    PROC StoreSlot_P02(num slot, num subType, num toolSel, num lenMM,
                       robtarget arcStart, robtarget arcEnd, robtarget approach, robtarget retract, robtarget trans)
        IF slot = 1 THEN
            P02W01_SubType := subType;
            P02W01_ToolSel := toolSel;
            P02W01_LenMM := lenMM;
            P02W01_ArcStart := arcStart;
            P02W01_ArcEnd := arcEnd;
            P02W01_Approach := approach;
            P02W01_Retract := retract;
            P02W01_Trans := trans;
            P02W01_Used := TRUE;
        ELSEIF slot = 2 THEN
            P02W02_SubType := subType;
            P02W02_ToolSel := toolSel;
            P02W02_LenMM := lenMM;
            P02W02_ArcStart := arcStart;
            P02W02_ArcEnd := arcEnd;
            P02W02_Approach := approach;
            P02W02_Retract := retract;
            P02W02_Trans := trans;
            P02W02_Used := TRUE;
        ELSEIF slot = 3 THEN
            P02W03_SubType := subType;
            P02W03_ToolSel := toolSel;
            P02W03_LenMM := lenMM;
            P02W03_ArcStart := arcStart;
            P02W03_ArcEnd := arcEnd;
            P02W03_Approach := approach;
            P02W03_Retract := retract;
            P02W03_Trans := trans;
            P02W03_Used := TRUE;
        ELSEIF slot = 4 THEN
            P02W04_SubType := subType;
            P02W04_ToolSel := toolSel;
            P02W04_LenMM := lenMM;
            P02W04_ArcStart := arcStart;
            P02W04_ArcEnd := arcEnd;
            P02W04_Approach := approach;
            P02W04_Retract := retract;
            P02W04_Trans := trans;
            P02W04_Used := TRUE;
        ELSEIF slot = 5 THEN
            P02W05_SubType := subType;
            P02W05_ToolSel := toolSel;
            P02W05_LenMM := lenMM;
            P02W05_ArcStart := arcStart;
            P02W05_ArcEnd := arcEnd;
            P02W05_Approach := approach;
            P02W05_Retract := retract;
            P02W05_Trans := trans;
            P02W05_Used := TRUE;
        ELSEIF slot = 6 THEN
            P02W06_SubType := subType;
            P02W06_ToolSel := toolSel;
            P02W06_LenMM := lenMM;
            P02W06_ArcStart := arcStart;
            P02W06_ArcEnd := arcEnd;
            P02W06_Approach := approach;
            P02W06_Retract := retract;
            P02W06_Trans := trans;
            P02W06_Used := TRUE;
        ELSEIF slot = 7 THEN
            P02W07_SubType := subType;
            P02W07_ToolSel := toolSel;
            P02W07_LenMM := lenMM;
            P02W07_ArcStart := arcStart;
            P02W07_ArcEnd := arcEnd;
            P02W07_Approach := approach;
            P02W07_Retract := retract;
            P02W07_Trans := trans;
            P02W07_Used := TRUE;
        ELSEIF slot = 8 THEN
            P02W08_SubType := subType;
            P02W08_ToolSel := toolSel;
            P02W08_LenMM := lenMM;
            P02W08_ArcStart := arcStart;
            P02W08_ArcEnd := arcEnd;
            P02W08_Approach := approach;
            P02W08_Retract := retract;
            P02W08_Trans := trans;
            P02W08_Used := TRUE;
        ELSEIF slot = 9 THEN
            P02W09_SubType := subType;
            P02W09_ToolSel := toolSel;
            P02W09_LenMM := lenMM;
            P02W09_ArcStart := arcStart;
            P02W09_ArcEnd := arcEnd;
            P02W09_Approach := approach;
            P02W09_Retract := retract;
            P02W09_Trans := trans;
            P02W09_Used := TRUE;
        ELSEIF slot = 10 THEN
            P02W10_SubType := subType;
            P02W10_ToolSel := toolSel;
            P02W10_LenMM := lenMM;
            P02W10_ArcStart := arcStart;
            P02W10_ArcEnd := arcEnd;
            P02W10_Approach := approach;
            P02W10_Retract := retract;
            P02W10_Trans := trans;
            P02W10_Used := TRUE;
        ELSEIF slot = 11 THEN
            P02W11_SubType := subType;
            P02W11_ToolSel := toolSel;
            P02W11_LenMM := lenMM;
            P02W11_ArcStart := arcStart;
            P02W11_ArcEnd := arcEnd;
            P02W11_Approach := approach;
            P02W11_Retract := retract;
            P02W11_Trans := trans;
            P02W11_Used := TRUE;
        ELSEIF slot = 12 THEN
            P02W12_SubType := subType;
            P02W12_ToolSel := toolSel;
            P02W12_LenMM := lenMM;
            P02W12_ArcStart := arcStart;
            P02W12_ArcEnd := arcEnd;
            P02W12_Approach := approach;
            P02W12_Retract := retract;
            P02W12_Trans := trans;
            P02W12_Used := TRUE;
        ELSEIF slot = 13 THEN
            P02W13_SubType := subType;
            P02W13_ToolSel := toolSel;
            P02W13_LenMM := lenMM;
            P02W13_ArcStart := arcStart;
            P02W13_ArcEnd := arcEnd;
            P02W13_Approach := approach;
            P02W13_Retract := retract;
            P02W13_Trans := trans;
            P02W13_Used := TRUE;
        ELSEIF slot = 14 THEN
            P02W14_SubType := subType;
            P02W14_ToolSel := toolSel;
            P02W14_LenMM := lenMM;
            P02W14_ArcStart := arcStart;
            P02W14_ArcEnd := arcEnd;
            P02W14_Approach := approach;
            P02W14_Retract := retract;
            P02W14_Trans := trans;
            P02W14_Used := TRUE;
        ELSEIF slot = 15 THEN
            P02W15_SubType := subType;
            P02W15_ToolSel := toolSel;
            P02W15_LenMM := lenMM;
            P02W15_ArcStart := arcStart;
            P02W15_ArcEnd := arcEnd;
            P02W15_Approach := approach;
            P02W15_Retract := retract;
            P02W15_Trans := trans;
            P02W15_Used := TRUE;
        ELSEIF slot = 16 THEN
            P02W16_SubType := subType;
            P02W16_ToolSel := toolSel;
            P02W16_LenMM := lenMM;
            P02W16_ArcStart := arcStart;
            P02W16_ArcEnd := arcEnd;
            P02W16_Approach := approach;
            P02W16_Retract := retract;
            P02W16_Trans := trans;
            P02W16_Used := TRUE;
        ELSEIF slot = 17 THEN
            P02W17_SubType := subType;
            P02W17_ToolSel := toolSel;
            P02W17_LenMM := lenMM;
            P02W17_ArcStart := arcStart;
            P02W17_ArcEnd := arcEnd;
            P02W17_Approach := approach;
            P02W17_Retract := retract;
            P02W17_Trans := trans;
            P02W17_Used := TRUE;
        ELSEIF slot = 18 THEN
            P02W18_SubType := subType;
            P02W18_ToolSel := toolSel;
            P02W18_LenMM := lenMM;
            P02W18_ArcStart := arcStart;
            P02W18_ArcEnd := arcEnd;
            P02W18_Approach := approach;
            P02W18_Retract := retract;
            P02W18_Trans := trans;
            P02W18_Used := TRUE;
        ELSEIF slot = 19 THEN
            P02W19_SubType := subType;
            P02W19_ToolSel := toolSel;
            P02W19_LenMM := lenMM;
            P02W19_ArcStart := arcStart;
            P02W19_ArcEnd := arcEnd;
            P02W19_Approach := approach;
            P02W19_Retract := retract;
            P02W19_Trans := trans;
            P02W19_Used := TRUE;
        ELSEIF slot = 20 THEN
            P02W20_SubType := subType;
            P02W20_ToolSel := toolSel;
            P02W20_LenMM := lenMM;
            P02W20_ArcStart := arcStart;
            P02W20_ArcEnd := arcEnd;
            P02W20_Approach := approach;
            P02W20_Retract := retract;
            P02W20_Trans := trans;
            P02W20_Used := TRUE;
        ELSEIF slot = 21 THEN
            P02W21_SubType := subType;
            P02W21_ToolSel := toolSel;
            P02W21_LenMM := lenMM;
            P02W21_ArcStart := arcStart;
            P02W21_ArcEnd := arcEnd;
            P02W21_Approach := approach;
            P02W21_Retract := retract;
            P02W21_Trans := trans;
            P02W21_Used := TRUE;
        ELSEIF slot = 22 THEN
            P02W22_SubType := subType;
            P02W22_ToolSel := toolSel;
            P02W22_LenMM := lenMM;
            P02W22_ArcStart := arcStart;
            P02W22_ArcEnd := arcEnd;
            P02W22_Approach := approach;
            P02W22_Retract := retract;
            P02W22_Trans := trans;
            P02W22_Used := TRUE;
        ELSEIF slot = 23 THEN
            P02W23_SubType := subType;
            P02W23_ToolSel := toolSel;
            P02W23_LenMM := lenMM;
            P02W23_ArcStart := arcStart;
            P02W23_ArcEnd := arcEnd;
            P02W23_Approach := approach;
            P02W23_Retract := retract;
            P02W23_Trans := trans;
            P02W23_Used := TRUE;
        ELSEIF slot = 24 THEN
            P02W24_SubType := subType;
            P02W24_ToolSel := toolSel;
            P02W24_LenMM := lenMM;
            P02W24_ArcStart := arcStart;
            P02W24_ArcEnd := arcEnd;
            P02W24_Approach := approach;
            P02W24_Retract := retract;
            P02W24_Trans := trans;
            P02W24_Used := TRUE;
        ELSEIF slot = 25 THEN
            P02W25_SubType := subType;
            P02W25_ToolSel := toolSel;
            P02W25_LenMM := lenMM;
            P02W25_ArcStart := arcStart;
            P02W25_ArcEnd := arcEnd;
            P02W25_Approach := approach;
            P02W25_Retract := retract;
            P02W25_Trans := trans;
            P02W25_Used := TRUE;
        ELSEIF slot = 26 THEN
            P02W26_SubType := subType;
            P02W26_ToolSel := toolSel;
            P02W26_LenMM := lenMM;
            P02W26_ArcStart := arcStart;
            P02W26_ArcEnd := arcEnd;
            P02W26_Approach := approach;
            P02W26_Retract := retract;
            P02W26_Trans := trans;
            P02W26_Used := TRUE;
        ELSEIF slot = 27 THEN
            P02W27_SubType := subType;
            P02W27_ToolSel := toolSel;
            P02W27_LenMM := lenMM;
            P02W27_ArcStart := arcStart;
            P02W27_ArcEnd := arcEnd;
            P02W27_Approach := approach;
            P02W27_Retract := retract;
            P02W27_Trans := trans;
            P02W27_Used := TRUE;
        ELSEIF slot = 28 THEN
            P02W28_SubType := subType;
            P02W28_ToolSel := toolSel;
            P02W28_LenMM := lenMM;
            P02W28_ArcStart := arcStart;
            P02W28_ArcEnd := arcEnd;
            P02W28_Approach := approach;
            P02W28_Retract := retract;
            P02W28_Trans := trans;
            P02W28_Used := TRUE;
        ELSEIF slot = 29 THEN
            P02W29_SubType := subType;
            P02W29_ToolSel := toolSel;
            P02W29_LenMM := lenMM;
            P02W29_ArcStart := arcStart;
            P02W29_ArcEnd := arcEnd;
            P02W29_Approach := approach;
            P02W29_Retract := retract;
            P02W29_Trans := trans;
            P02W29_Used := TRUE;
        ELSEIF slot = 30 THEN
            P02W30_SubType := subType;
            P02W30_ToolSel := toolSel;
            P02W30_LenMM := lenMM;
            P02W30_ArcStart := arcStart;
            P02W30_ArcEnd := arcEnd;
            P02W30_Approach := approach;
            P02W30_Retract := retract;
            P02W30_Trans := trans;
            P02W30_Used := TRUE;
        ELSE
            TPWrite "Invalid weld slot.";
        ENDIF
    ENDPROC

    PROC LoadSlot_P02(num slot, VAR bool used, VAR num subType, VAR num toolSel, VAR num lenMM,
                       VAR robtarget arcStart, VAR robtarget arcEnd, VAR robtarget approach, VAR robtarget retract, VAR robtarget trans)
        IF slot = 1 THEN
            used := P02W01_Used;
            subType := P02W01_SubType;
            toolSel := P02W01_ToolSel;
            lenMM := P02W01_LenMM;
            arcStart := P02W01_ArcStart;
            arcEnd := P02W01_ArcEnd;
            approach := P02W01_Approach;
            retract := P02W01_Retract;
            trans := P02W01_Trans;
        ELSEIF slot = 2 THEN
            used := P02W02_Used;
            subType := P02W02_SubType;
            toolSel := P02W02_ToolSel;
            lenMM := P02W02_LenMM;
            arcStart := P02W02_ArcStart;
            arcEnd := P02W02_ArcEnd;
            approach := P02W02_Approach;
            retract := P02W02_Retract;
            trans := P02W02_Trans;
        ELSEIF slot = 3 THEN
            used := P02W03_Used;
            subType := P02W03_SubType;
            toolSel := P02W03_ToolSel;
            lenMM := P02W03_LenMM;
            arcStart := P02W03_ArcStart;
            arcEnd := P02W03_ArcEnd;
            approach := P02W03_Approach;
            retract := P02W03_Retract;
            trans := P02W03_Trans;
        ELSEIF slot = 4 THEN
            used := P02W04_Used;
            subType := P02W04_SubType;
            toolSel := P02W04_ToolSel;
            lenMM := P02W04_LenMM;
            arcStart := P02W04_ArcStart;
            arcEnd := P02W04_ArcEnd;
            approach := P02W04_Approach;
            retract := P02W04_Retract;
            trans := P02W04_Trans;
        ELSEIF slot = 5 THEN
            used := P02W05_Used;
            subType := P02W05_SubType;
            toolSel := P02W05_ToolSel;
            lenMM := P02W05_LenMM;
            arcStart := P02W05_ArcStart;
            arcEnd := P02W05_ArcEnd;
            approach := P02W05_Approach;
            retract := P02W05_Retract;
            trans := P02W05_Trans;
        ELSEIF slot = 6 THEN
            used := P02W06_Used;
            subType := P02W06_SubType;
            toolSel := P02W06_ToolSel;
            lenMM := P02W06_LenMM;
            arcStart := P02W06_ArcStart;
            arcEnd := P02W06_ArcEnd;
            approach := P02W06_Approach;
            retract := P02W06_Retract;
            trans := P02W06_Trans;
        ELSEIF slot = 7 THEN
            used := P02W07_Used;
            subType := P02W07_SubType;
            toolSel := P02W07_ToolSel;
            lenMM := P02W07_LenMM;
            arcStart := P02W07_ArcStart;
            arcEnd := P02W07_ArcEnd;
            approach := P02W07_Approach;
            retract := P02W07_Retract;
            trans := P02W07_Trans;
        ELSEIF slot = 8 THEN
            used := P02W08_Used;
            subType := P02W08_SubType;
            toolSel := P02W08_ToolSel;
            lenMM := P02W08_LenMM;
            arcStart := P02W08_ArcStart;
            arcEnd := P02W08_ArcEnd;
            approach := P02W08_Approach;
            retract := P02W08_Retract;
            trans := P02W08_Trans;
        ELSEIF slot = 9 THEN
            used := P02W09_Used;
            subType := P02W09_SubType;
            toolSel := P02W09_ToolSel;
            lenMM := P02W09_LenMM;
            arcStart := P02W09_ArcStart;
            arcEnd := P02W09_ArcEnd;
            approach := P02W09_Approach;
            retract := P02W09_Retract;
            trans := P02W09_Trans;
        ELSEIF slot = 10 THEN
            used := P02W10_Used;
            subType := P02W10_SubType;
            toolSel := P02W10_ToolSel;
            lenMM := P02W10_LenMM;
            arcStart := P02W10_ArcStart;
            arcEnd := P02W10_ArcEnd;
            approach := P02W10_Approach;
            retract := P02W10_Retract;
            trans := P02W10_Trans;
        ELSEIF slot = 11 THEN
            used := P02W11_Used;
            subType := P02W11_SubType;
            toolSel := P02W11_ToolSel;
            lenMM := P02W11_LenMM;
            arcStart := P02W11_ArcStart;
            arcEnd := P02W11_ArcEnd;
            approach := P02W11_Approach;
            retract := P02W11_Retract;
            trans := P02W11_Trans;
        ELSEIF slot = 12 THEN
            used := P02W12_Used;
            subType := P02W12_SubType;
            toolSel := P02W12_ToolSel;
            lenMM := P02W12_LenMM;
            arcStart := P02W12_ArcStart;
            arcEnd := P02W12_ArcEnd;
            approach := P02W12_Approach;
            retract := P02W12_Retract;
            trans := P02W12_Trans;
        ELSEIF slot = 13 THEN
            used := P02W13_Used;
            subType := P02W13_SubType;
            toolSel := P02W13_ToolSel;
            lenMM := P02W13_LenMM;
            arcStart := P02W13_ArcStart;
            arcEnd := P02W13_ArcEnd;
            approach := P02W13_Approach;
            retract := P02W13_Retract;
            trans := P02W13_Trans;
        ELSEIF slot = 14 THEN
            used := P02W14_Used;
            subType := P02W14_SubType;
            toolSel := P02W14_ToolSel;
            lenMM := P02W14_LenMM;
            arcStart := P02W14_ArcStart;
            arcEnd := P02W14_ArcEnd;
            approach := P02W14_Approach;
            retract := P02W14_Retract;
            trans := P02W14_Trans;
        ELSEIF slot = 15 THEN
            used := P02W15_Used;
            subType := P02W15_SubType;
            toolSel := P02W15_ToolSel;
            lenMM := P02W15_LenMM;
            arcStart := P02W15_ArcStart;
            arcEnd := P02W15_ArcEnd;
            approach := P02W15_Approach;
            retract := P02W15_Retract;
            trans := P02W15_Trans;
        ELSEIF slot = 16 THEN
            used := P02W16_Used;
            subType := P02W16_SubType;
            toolSel := P02W16_ToolSel;
            lenMM := P02W16_LenMM;
            arcStart := P02W16_ArcStart;
            arcEnd := P02W16_ArcEnd;
            approach := P02W16_Approach;
            retract := P02W16_Retract;
            trans := P02W16_Trans;
        ELSEIF slot = 17 THEN
            used := P02W17_Used;
            subType := P02W17_SubType;
            toolSel := P02W17_ToolSel;
            lenMM := P02W17_LenMM;
            arcStart := P02W17_ArcStart;
            arcEnd := P02W17_ArcEnd;
            approach := P02W17_Approach;
            retract := P02W17_Retract;
            trans := P02W17_Trans;
        ELSEIF slot = 18 THEN
            used := P02W18_Used;
            subType := P02W18_SubType;
            toolSel := P02W18_ToolSel;
            lenMM := P02W18_LenMM;
            arcStart := P02W18_ArcStart;
            arcEnd := P02W18_ArcEnd;
            approach := P02W18_Approach;
            retract := P02W18_Retract;
            trans := P02W18_Trans;
        ELSEIF slot = 19 THEN
            used := P02W19_Used;
            subType := P02W19_SubType;
            toolSel := P02W19_ToolSel;
            lenMM := P02W19_LenMM;
            arcStart := P02W19_ArcStart;
            arcEnd := P02W19_ArcEnd;
            approach := P02W19_Approach;
            retract := P02W19_Retract;
            trans := P02W19_Trans;
        ELSEIF slot = 20 THEN
            used := P02W20_Used;
            subType := P02W20_SubType;
            toolSel := P02W20_ToolSel;
            lenMM := P02W20_LenMM;
            arcStart := P02W20_ArcStart;
            arcEnd := P02W20_ArcEnd;
            approach := P02W20_Approach;
            retract := P02W20_Retract;
            trans := P02W20_Trans;
        ELSEIF slot = 21 THEN
            used := P02W21_Used;
            subType := P02W21_SubType;
            toolSel := P02W21_ToolSel;
            lenMM := P02W21_LenMM;
            arcStart := P02W21_ArcStart;
            arcEnd := P02W21_ArcEnd;
            approach := P02W21_Approach;
            retract := P02W21_Retract;
            trans := P02W21_Trans;
        ELSEIF slot = 22 THEN
            used := P02W22_Used;
            subType := P02W22_SubType;
            toolSel := P02W22_ToolSel;
            lenMM := P02W22_LenMM;
            arcStart := P02W22_ArcStart;
            arcEnd := P02W22_ArcEnd;
            approach := P02W22_Approach;
            retract := P02W22_Retract;
            trans := P02W22_Trans;
        ELSEIF slot = 23 THEN
            used := P02W23_Used;
            subType := P02W23_SubType;
            toolSel := P02W23_ToolSel;
            lenMM := P02W23_LenMM;
            arcStart := P02W23_ArcStart;
            arcEnd := P02W23_ArcEnd;
            approach := P02W23_Approach;
            retract := P02W23_Retract;
            trans := P02W23_Trans;
        ELSEIF slot = 24 THEN
            used := P02W24_Used;
            subType := P02W24_SubType;
            toolSel := P02W24_ToolSel;
            lenMM := P02W24_LenMM;
            arcStart := P02W24_ArcStart;
            arcEnd := P02W24_ArcEnd;
            approach := P02W24_Approach;
            retract := P02W24_Retract;
            trans := P02W24_Trans;
        ELSEIF slot = 25 THEN
            used := P02W25_Used;
            subType := P02W25_SubType;
            toolSel := P02W25_ToolSel;
            lenMM := P02W25_LenMM;
            arcStart := P02W25_ArcStart;
            arcEnd := P02W25_ArcEnd;
            approach := P02W25_Approach;
            retract := P02W25_Retract;
            trans := P02W25_Trans;
        ELSEIF slot = 26 THEN
            used := P02W26_Used;
            subType := P02W26_SubType;
            toolSel := P02W26_ToolSel;
            lenMM := P02W26_LenMM;
            arcStart := P02W26_ArcStart;
            arcEnd := P02W26_ArcEnd;
            approach := P02W26_Approach;
            retract := P02W26_Retract;
            trans := P02W26_Trans;
        ELSEIF slot = 27 THEN
            used := P02W27_Used;
            subType := P02W27_SubType;
            toolSel := P02W27_ToolSel;
            lenMM := P02W27_LenMM;
            arcStart := P02W27_ArcStart;
            arcEnd := P02W27_ArcEnd;
            approach := P02W27_Approach;
            retract := P02W27_Retract;
            trans := P02W27_Trans;
        ELSEIF slot = 28 THEN
            used := P02W28_Used;
            subType := P02W28_SubType;
            toolSel := P02W28_ToolSel;
            lenMM := P02W28_LenMM;
            arcStart := P02W28_ArcStart;
            arcEnd := P02W28_ArcEnd;
            approach := P02W28_Approach;
            retract := P02W28_Retract;
            trans := P02W28_Trans;
        ELSEIF slot = 29 THEN
            used := P02W29_Used;
            subType := P02W29_SubType;
            toolSel := P02W29_ToolSel;
            lenMM := P02W29_LenMM;
            arcStart := P02W29_ArcStart;
            arcEnd := P02W29_ArcEnd;
            approach := P02W29_Approach;
            retract := P02W29_Retract;
            trans := P02W29_Trans;
        ELSEIF slot = 30 THEN
            used := P02W30_Used;
            subType := P02W30_SubType;
            toolSel := P02W30_ToolSel;
            lenMM := P02W30_LenMM;
            arcStart := P02W30_ArcStart;
            arcEnd := P02W30_ArcEnd;
            approach := P02W30_Approach;
            retract := P02W30_Retract;
            trans := P02W30_Trans;
        ELSE
            used := FALSE;
        ENDIF
    ENDPROC

    PROC ClearSlot_P02(num slot)
        IF slot = 1 THEN
            P02W01_Used := FALSE;
            P02W01_SubType := 0;
            P02W01_ToolSel := 0;
            P02W01_LenMM := 0;
            P02W01_ArcStart := [[0,0,0],[1,0,0,0],[0,0,0,0],[9E9,9E9,9E9,9E9,9E9,9E9]];
            P02W01_ArcEnd := [[0,0,0],[1,0,0,0],[0,0,0,0],[9E9,9E9,9E9,9E9,9E9,9E9]];
            P02W01_Approach := [[0,0,0],[1,0,0,0],[0,0,0,0],[9E9,9E9,9E9,9E9,9E9,9E9]];
            P02W01_Retract := [[0,0,0],[1,0,0,0],[0,0,0,0],[9E9,9E9,9E9,9E9,9E9,9E9]];
            P02W01_Trans := [[0,0,0],[1,0,0,0],[0,0,0,0],[9E9,9E9,9E9,9E9,9E9,9E9]];
        ELSEIF slot = 2 THEN
            P02W02_Used := FALSE;
            P02W02_SubType := 0;
            P02W02_ToolSel := 0;
            P02W02_LenMM := 0;
            P02W02_ArcStart := [[0,0,0],[1,0,0,0],[0,0,0,0],[9E9,9E9,9E9,9E9,9E9,9E9]];
            P02W02_ArcEnd := [[0,0,0],[1,0,0,0],[0,0,0,0],[9E9,9E9,9E9,9E9,9E9,9E9]];
            P02W02_Approach := [[0,0,0],[1,0,0,0],[0,0,0,0],[9E9,9E9,9E9,9E9,9E9,9E9]];
            P02W02_Retract := [[0,0,0],[1,0,0,0],[0,0,0,0],[9E9,9E9,9E9,9E9,9E9,9E9]];
            P02W02_Trans := [[0,0,0],[1,0,0,0],[0,0,0,0],[9E9,9E9,9E9,9E9,9E9,9E9]];
        ELSEIF slot = 3 THEN
            P02W03_Used := FALSE;
            P02W03_SubType := 0;
            P02W03_ToolSel := 0;
            P02W03_LenMM := 0;
            P02W03_ArcStart := [[0,0,0],[1,0,0,0],[0,0,0,0],[9E9,9E9,9E9,9E9,9E9,9E9]];
            P02W03_ArcEnd := [[0,0,0],[1,0,0,0],[0,0,0,0],[9E9,9E9,9E9,9E9,9E9,9E9]];
            P02W03_Approach := [[0,0,0],[1,0,0,0],[0,0,0,0],[9E9,9E9,9E9,9E9,9E9,9E9]];
            P02W03_Retract := [[0,0,0],[1,0,0,0],[0,0,0,0],[9E9,9E9,9E9,9E9,9E9,9E9]];
            P02W03_Trans := [[0,0,0],[1,0,0,0],[0,0,0,0],[9E9,9E9,9E9,9E9,9E9,9E9]];
        ELSEIF slot = 4 THEN
            P02W04_Used := FALSE;
            P02W04_SubType := 0;
            P02W04_ToolSel := 0;
            P02W04_LenMM := 0;
            P02W04_ArcStart := [[0,0,0],[1,0,0,0],[0,0,0,0],[9E9,9E9,9E9,9E9,9E9,9E9]];
            P02W04_ArcEnd := [[0,0,0],[1,0,0,0],[0,0,0,0],[9E9,9E9,9E9,9E9,9E9,9E9]];
            P02W04_Approach := [[0,0,0],[1,0,0,0],[0,0,0,0],[9E9,9E9,9E9,9E9,9E9,9E9]];
            P02W04_Retract := [[0,0,0],[1,0,0,0],[0,0,0,0],[9E9,9E9,9E9,9E9,9E9,9E9]];
            P02W04_Trans := [[0,0,0],[1,0,0,0],[0,0,0,0],[9E9,9E9,9E9,9E9,9E9,9E9]];
        ELSEIF slot = 5 THEN
            P02W05_Used := FALSE;
            P02W05_SubType := 0;
            P02W05_ToolSel := 0;
            P02W05_LenMM := 0;
            P02W05_ArcStart := [[0,0,0],[1,0,0,0],[0,0,0,0],[9E9,9E9,9E9,9E9,9E9,9E9]];
            P02W05_ArcEnd := [[0,0,0],[1,0,0,0],[0,0,0,0],[9E9,9E9,9E9,9E9,9E9,9E9]];
            P02W05_Approach := [[0,0,0],[1,0,0,0],[0,0,0,0],[9E9,9E9,9E9,9E9,9E9,9E9]];
            P02W05_Retract := [[0,0,0],[1,0,0,0],[0,0,0,0],[9E9,9E9,9E9,9E9,9E9,9E9]];
            P02W05_Trans := [[0,0,0],[1,0,0,0],[0,0,0,0],[9E9,9E9,9E9,9E9,9E9,9E9]];
        ELSEIF slot = 6 THEN
            P02W06_Used := FALSE;
            P02W06_SubType := 0;
            P02W06_ToolSel := 0;
            P02W06_LenMM := 0;
            P02W06_ArcStart := [[0,0,0],[1,0,0,0],[0,0,0,0],[9E9,9E9,9E9,9E9,9E9,9E9]];
            P02W06_ArcEnd := [[0,0,0],[1,0,0,0],[0,0,0,0],[9E9,9E9,9E9,9E9,9E9,9E9]];
            P02W06_Approach := [[0,0,0],[1,0,0,0],[0,0,0,0],[9E9,9E9,9E9,9E9,9E9,9E9]];
            P02W06_Retract := [[0,0,0],[1,0,0,0],[0,0,0,0],[9E9,9E9,9E9,9E9,9E9,9E9]];
            P02W06_Trans := [[0,0,0],[1,0,0,0],[0,0,0,0],[9E9,9E9,9E9,9E9,9E9,9E9]];
        ELSEIF slot = 7 THEN
            P02W07_Used := FALSE;
            P02W07_SubType := 0;
            P02W07_ToolSel := 0;
            P02W07_LenMM := 0;
            P02W07_ArcStart := [[0,0,0],[1,0,0,0],[0,0,0,0],[9E9,9E9,9E9,9E9,9E9,9E9]];
            P02W07_ArcEnd := [[0,0,0],[1,0,0,0],[0,0,0,0],[9E9,9E9,9E9,9E9,9E9,9E9]];
            P02W07_Approach := [[0,0,0],[1,0,0,0],[0,0,0,0],[9E9,9E9,9E9,9E9,9E9,9E9]];
            P02W07_Retract := [[0,0,0],[1,0,0,0],[0,0,0,0],[9E9,9E9,9E9,9E9,9E9,9E9]];
            P02W07_Trans := [[0,0,0],[1,0,0,0],[0,0,0,0],[9E9,9E9,9E9,9E9,9E9,9E9]];
        ELSEIF slot = 8 THEN
            P02W08_Used := FALSE;
            P02W08_SubType := 0;
            P02W08_ToolSel := 0;
            P02W08_LenMM := 0;
            P02W08_ArcStart := [[0,0,0],[1,0,0,0],[0,0,0,0],[9E9,9E9,9E9,9E9,9E9,9E9]];
            P02W08_ArcEnd := [[0,0,0],[1,0,0,0],[0,0,0,0],[9E9,9E9,9E9,9E9,9E9,9E9]];
            P02W08_Approach := [[0,0,0],[1,0,0,0],[0,0,0,0],[9E9,9E9,9E9,9E9,9E9,9E9]];
            P02W08_Retract := [[0,0,0],[1,0,0,0],[0,0,0,0],[9E9,9E9,9E9,9E9,9E9,9E9]];
            P02W08_Trans := [[0,0,0],[1,0,0,0],[0,0,0,0],[9E9,9E9,9E9,9E9,9E9,9E9]];
        ELSEIF slot = 9 THEN
            P02W09_Used := FALSE;
            P02W09_SubType := 0;
            P02W09_ToolSel := 0;
            P02W09_LenMM := 0;
            P02W09_ArcStart := [[0,0,0],[1,0,0,0],[0,0,0,0],[9E9,9E9,9E9,9E9,9E9,9E9]];
            P02W09_ArcEnd := [[0,0,0],[1,0,0,0],[0,0,0,0],[9E9,9E9,9E9,9E9,9E9,9E9]];
            P02W09_Approach := [[0,0,0],[1,0,0,0],[0,0,0,0],[9E9,9E9,9E9,9E9,9E9,9E9]];
            P02W09_Retract := [[0,0,0],[1,0,0,0],[0,0,0,0],[9E9,9E9,9E9,9E9,9E9,9E9]];
            P02W09_Trans := [[0,0,0],[1,0,0,0],[0,0,0,0],[9E9,9E9,9E9,9E9,9E9,9E9]];
        ELSEIF slot = 10 THEN
            P02W10_Used := FALSE;
            P02W10_SubType := 0;
            P02W10_ToolSel := 0;
            P02W10_LenMM := 0;
            P02W10_ArcStart := [[0,0,0],[1,0,0,0],[0,0,0,0],[9E9,9E9,9E9,9E9,9E9,9E9]];
            P02W10_ArcEnd := [[0,0,0],[1,0,0,0],[0,0,0,0],[9E9,9E9,9E9,9E9,9E9,9E9]];
            P02W10_Approach := [[0,0,0],[1,0,0,0],[0,0,0,0],[9E9,9E9,9E9,9E9,9E9,9E9]];
            P02W10_Retract := [[0,0,0],[1,0,0,0],[0,0,0,0],[9E9,9E9,9E9,9E9,9E9,9E9]];
            P02W10_Trans := [[0,0,0],[1,0,0,0],[0,0,0,0],[9E9,9E9,9E9,9E9,9E9,9E9]];
        ELSEIF slot = 11 THEN
            P02W11_Used := FALSE;
            P02W11_SubType := 0;
            P02W11_ToolSel := 0;
            P02W11_LenMM := 0;
            P02W11_ArcStart := [[0,0,0],[1,0,0,0],[0,0,0,0],[9E9,9E9,9E9,9E9,9E9,9E9]];
            P02W11_ArcEnd := [[0,0,0],[1,0,0,0],[0,0,0,0],[9E9,9E9,9E9,9E9,9E9,9E9]];
            P02W11_Approach := [[0,0,0],[1,0,0,0],[0,0,0,0],[9E9,9E9,9E9,9E9,9E9,9E9]];
            P02W11_Retract := [[0,0,0],[1,0,0,0],[0,0,0,0],[9E9,9E9,9E9,9E9,9E9,9E9]];
            P02W11_Trans := [[0,0,0],[1,0,0,0],[0,0,0,0],[9E9,9E9,9E9,9E9,9E9,9E9]];
        ELSEIF slot = 12 THEN
            P02W12_Used := FALSE;
            P02W12_SubType := 0;
            P02W12_ToolSel := 0;
            P02W12_LenMM := 0;
            P02W12_ArcStart := [[0,0,0],[1,0,0,0],[0,0,0,0],[9E9,9E9,9E9,9E9,9E9,9E9]];
            P02W12_ArcEnd := [[0,0,0],[1,0,0,0],[0,0,0,0],[9E9,9E9,9E9,9E9,9E9,9E9]];
            P02W12_Approach := [[0,0,0],[1,0,0,0],[0,0,0,0],[9E9,9E9,9E9,9E9,9E9,9E9]];
            P02W12_Retract := [[0,0,0],[1,0,0,0],[0,0,0,0],[9E9,9E9,9E9,9E9,9E9,9E9]];
            P02W12_Trans := [[0,0,0],[1,0,0,0],[0,0,0,0],[9E9,9E9,9E9,9E9,9E9,9E9]];
        ELSEIF slot = 13 THEN
            P02W13_Used := FALSE;
            P02W13_SubType := 0;
            P02W13_ToolSel := 0;
            P02W13_LenMM := 0;
            P02W13_ArcStart := [[0,0,0],[1,0,0,0],[0,0,0,0],[9E9,9E9,9E9,9E9,9E9,9E9]];
            P02W13_ArcEnd := [[0,0,0],[1,0,0,0],[0,0,0,0],[9E9,9E9,9E9,9E9,9E9,9E9]];
            P02W13_Approach := [[0,0,0],[1,0,0,0],[0,0,0,0],[9E9,9E9,9E9,9E9,9E9,9E9]];
            P02W13_Retract := [[0,0,0],[1,0,0,0],[0,0,0,0],[9E9,9E9,9E9,9E9,9E9,9E9]];
            P02W13_Trans := [[0,0,0],[1,0,0,0],[0,0,0,0],[9E9,9E9,9E9,9E9,9E9,9E9]];
        ELSEIF slot = 14 THEN
            P02W14_Used := FALSE;
            P02W14_SubType := 0;
            P02W14_ToolSel := 0;
            P02W14_LenMM := 0;
            P02W14_ArcStart := [[0,0,0],[1,0,0,0],[0,0,0,0],[9E9,9E9,9E9,9E9,9E9,9E9]];
            P02W14_ArcEnd := [[0,0,0],[1,0,0,0],[0,0,0,0],[9E9,9E9,9E9,9E9,9E9,9E9]];
            P02W14_Approach := [[0,0,0],[1,0,0,0],[0,0,0,0],[9E9,9E9,9E9,9E9,9E9,9E9]];
            P02W14_Retract := [[0,0,0],[1,0,0,0],[0,0,0,0],[9E9,9E9,9E9,9E9,9E9,9E9]];
            P02W14_Trans := [[0,0,0],[1,0,0,0],[0,0,0,0],[9E9,9E9,9E9,9E9,9E9,9E9]];
        ELSEIF slot = 15 THEN
            P02W15_Used := FALSE;
            P02W15_SubType := 0;
            P02W15_ToolSel := 0;
            P02W15_LenMM := 0;
            P02W15_ArcStart := [[0,0,0],[1,0,0,0],[0,0,0,0],[9E9,9E9,9E9,9E9,9E9,9E9]];
            P02W15_ArcEnd := [[0,0,0],[1,0,0,0],[0,0,0,0],[9E9,9E9,9E9,9E9,9E9,9E9]];
            P02W15_Approach := [[0,0,0],[1,0,0,0],[0,0,0,0],[9E9,9E9,9E9,9E9,9E9,9E9]];
            P02W15_Retract := [[0,0,0],[1,0,0,0],[0,0,0,0],[9E9,9E9,9E9,9E9,9E9,9E9]];
            P02W15_Trans := [[0,0,0],[1,0,0,0],[0,0,0,0],[9E9,9E9,9E9,9E9,9E9,9E9]];
        ELSEIF slot = 16 THEN
            P02W16_Used := FALSE;
            P02W16_SubType := 0;
            P02W16_ToolSel := 0;
            P02W16_LenMM := 0;
            P02W16_ArcStart := [[0,0,0],[1,0,0,0],[0,0,0,0],[9E9,9E9,9E9,9E9,9E9,9E9]];
            P02W16_ArcEnd := [[0,0,0],[1,0,0,0],[0,0,0,0],[9E9,9E9,9E9,9E9,9E9,9E9]];
            P02W16_Approach := [[0,0,0],[1,0,0,0],[0,0,0,0],[9E9,9E9,9E9,9E9,9E9,9E9]];
            P02W16_Retract := [[0,0,0],[1,0,0,0],[0,0,0,0],[9E9,9E9,9E9,9E9,9E9,9E9]];
            P02W16_Trans := [[0,0,0],[1,0,0,0],[0,0,0,0],[9E9,9E9,9E9,9E9,9E9,9E9]];
        ELSEIF slot = 17 THEN
            P02W17_Used := FALSE;
            P02W17_SubType := 0;
            P02W17_ToolSel := 0;
            P02W17_LenMM := 0;
            P02W17_ArcStart := [[0,0,0],[1,0,0,0],[0,0,0,0],[9E9,9E9,9E9,9E9,9E9,9E9]];
            P02W17_ArcEnd := [[0,0,0],[1,0,0,0],[0,0,0,0],[9E9,9E9,9E9,9E9,9E9,9E9]];
            P02W17_Approach := [[0,0,0],[1,0,0,0],[0,0,0,0],[9E9,9E9,9E9,9E9,9E9,9E9]];
            P02W17_Retract := [[0,0,0],[1,0,0,0],[0,0,0,0],[9E9,9E9,9E9,9E9,9E9,9E9]];
            P02W17_Trans := [[0,0,0],[1,0,0,0],[0,0,0,0],[9E9,9E9,9E9,9E9,9E9,9E9]];
        ELSEIF slot = 18 THEN
            P02W18_Used := FALSE;
            P02W18_SubType := 0;
            P02W18_ToolSel := 0;
            P02W18_LenMM := 0;
            P02W18_ArcStart := [[0,0,0],[1,0,0,0],[0,0,0,0],[9E9,9E9,9E9,9E9,9E9,9E9]];
            P02W18_ArcEnd := [[0,0,0],[1,0,0,0],[0,0,0,0],[9E9,9E9,9E9,9E9,9E9,9E9]];
            P02W18_Approach := [[0,0,0],[1,0,0,0],[0,0,0,0],[9E9,9E9,9E9,9E9,9E9,9E9]];
            P02W18_Retract := [[0,0,0],[1,0,0,0],[0,0,0,0],[9E9,9E9,9E9,9E9,9E9,9E9]];
            P02W18_Trans := [[0,0,0],[1,0,0,0],[0,0,0,0],[9E9,9E9,9E9,9E9,9E9,9E9]];
        ELSEIF slot = 19 THEN
            P02W19_Used := FALSE;
            P02W19_SubType := 0;
            P02W19_ToolSel := 0;
            P02W19_LenMM := 0;
            P02W19_ArcStart := [[0,0,0],[1,0,0,0],[0,0,0,0],[9E9,9E9,9E9,9E9,9E9,9E9]];
            P02W19_ArcEnd := [[0,0,0],[1,0,0,0],[0,0,0,0],[9E9,9E9,9E9,9E9,9E9,9E9]];
            P02W19_Approach := [[0,0,0],[1,0,0,0],[0,0,0,0],[9E9,9E9,9E9,9E9,9E9,9E9]];
            P02W19_Retract := [[0,0,0],[1,0,0,0],[0,0,0,0],[9E9,9E9,9E9,9E9,9E9,9E9]];
            P02W19_Trans := [[0,0,0],[1,0,0,0],[0,0,0,0],[9E9,9E9,9E9,9E9,9E9,9E9]];
        ELSEIF slot = 20 THEN
            P02W20_Used := FALSE;
            P02W20_SubType := 0;
            P02W20_ToolSel := 0;
            P02W20_LenMM := 0;
            P02W20_ArcStart := [[0,0,0],[1,0,0,0],[0,0,0,0],[9E9,9E9,9E9,9E9,9E9,9E9]];
            P02W20_ArcEnd := [[0,0,0],[1,0,0,0],[0,0,0,0],[9E9,9E9,9E9,9E9,9E9,9E9]];
            P02W20_Approach := [[0,0,0],[1,0,0,0],[0,0,0,0],[9E9,9E9,9E9,9E9,9E9,9E9]];
            P02W20_Retract := [[0,0,0],[1,0,0,0],[0,0,0,0],[9E9,9E9,9E9,9E9,9E9,9E9]];
            P02W20_Trans := [[0,0,0],[1,0,0,0],[0,0,0,0],[9E9,9E9,9E9,9E9,9E9,9E9]];
        ELSEIF slot = 21 THEN
            P02W21_Used := FALSE;
            P02W21_SubType := 0;
            P02W21_ToolSel := 0;
            P02W21_LenMM := 0;
            P02W21_ArcStart := [[0,0,0],[1,0,0,0],[0,0,0,0],[9E9,9E9,9E9,9E9,9E9,9E9]];
            P02W21_ArcEnd := [[0,0,0],[1,0,0,0],[0,0,0,0],[9E9,9E9,9E9,9E9,9E9,9E9]];
            P02W21_Approach := [[0,0,0],[1,0,0,0],[0,0,0,0],[9E9,9E9,9E9,9E9,9E9,9E9]];
            P02W21_Retract := [[0,0,0],[1,0,0,0],[0,0,0,0],[9E9,9E9,9E9,9E9,9E9,9E9]];
            P02W21_Trans := [[0,0,0],[1,0,0,0],[0,0,0,0],[9E9,9E9,9E9,9E9,9E9,9E9]];
        ELSEIF slot = 22 THEN
            P02W22_Used := FALSE;
            P02W22_SubType := 0;
            P02W22_ToolSel := 0;
            P02W22_LenMM := 0;
            P02W22_ArcStart := [[0,0,0],[1,0,0,0],[0,0,0,0],[9E9,9E9,9E9,9E9,9E9,9E9]];
            P02W22_ArcEnd := [[0,0,0],[1,0,0,0],[0,0,0,0],[9E9,9E9,9E9,9E9,9E9,9E9]];
            P02W22_Approach := [[0,0,0],[1,0,0,0],[0,0,0,0],[9E9,9E9,9E9,9E9,9E9,9E9]];
            P02W22_Retract := [[0,0,0],[1,0,0,0],[0,0,0,0],[9E9,9E9,9E9,9E9,9E9,9E9]];
            P02W22_Trans := [[0,0,0],[1,0,0,0],[0,0,0,0],[9E9,9E9,9E9,9E9,9E9,9E9]];
        ELSEIF slot = 23 THEN
            P02W23_Used := FALSE;
            P02W23_SubType := 0;
            P02W23_ToolSel := 0;
            P02W23_LenMM := 0;
            P02W23_ArcStart := [[0,0,0],[1,0,0,0],[0,0,0,0],[9E9,9E9,9E9,9E9,9E9,9E9]];
            P02W23_ArcEnd := [[0,0,0],[1,0,0,0],[0,0,0,0],[9E9,9E9,9E9,9E9,9E9,9E9]];
            P02W23_Approach := [[0,0,0],[1,0,0,0],[0,0,0,0],[9E9,9E9,9E9,9E9,9E9,9E9]];
            P02W23_Retract := [[0,0,0],[1,0,0,0],[0,0,0,0],[9E9,9E9,9E9,9E9,9E9,9E9]];
            P02W23_Trans := [[0,0,0],[1,0,0,0],[0,0,0,0],[9E9,9E9,9E9,9E9,9E9,9E9]];
        ELSEIF slot = 24 THEN
            P02W24_Used := FALSE;
            P02W24_SubType := 0;
            P02W24_ToolSel := 0;
            P02W24_LenMM := 0;
            P02W24_ArcStart := [[0,0,0],[1,0,0,0],[0,0,0,0],[9E9,9E9,9E9,9E9,9E9,9E9]];
            P02W24_ArcEnd := [[0,0,0],[1,0,0,0],[0,0,0,0],[9E9,9E9,9E9,9E9,9E9,9E9]];
            P02W24_Approach := [[0,0,0],[1,0,0,0],[0,0,0,0],[9E9,9E9,9E9,9E9,9E9,9E9]];
            P02W24_Retract := [[0,0,0],[1,0,0,0],[0,0,0,0],[9E9,9E9,9E9,9E9,9E9,9E9]];
            P02W24_Trans := [[0,0,0],[1,0,0,0],[0,0,0,0],[9E9,9E9,9E9,9E9,9E9,9E9]];
        ELSEIF slot = 25 THEN
            P02W25_Used := FALSE;
            P02W25_SubType := 0;
            P02W25_ToolSel := 0;
            P02W25_LenMM := 0;
            P02W25_ArcStart := [[0,0,0],[1,0,0,0],[0,0,0,0],[9E9,9E9,9E9,9E9,9E9,9E9]];
            P02W25_ArcEnd := [[0,0,0],[1,0,0,0],[0,0,0,0],[9E9,9E9,9E9,9E9,9E9,9E9]];
            P02W25_Approach := [[0,0,0],[1,0,0,0],[0,0,0,0],[9E9,9E9,9E9,9E9,9E9,9E9]];
            P02W25_Retract := [[0,0,0],[1,0,0,0],[0,0,0,0],[9E9,9E9,9E9,9E9,9E9,9E9]];
            P02W25_Trans := [[0,0,0],[1,0,0,0],[0,0,0,0],[9E9,9E9,9E9,9E9,9E9,9E9]];
        ELSEIF slot = 26 THEN
            P02W26_Used := FALSE;
            P02W26_SubType := 0;
            P02W26_ToolSel := 0;
            P02W26_LenMM := 0;
            P02W26_ArcStart := [[0,0,0],[1,0,0,0],[0,0,0,0],[9E9,9E9,9E9,9E9,9E9,9E9]];
            P02W26_ArcEnd := [[0,0,0],[1,0,0,0],[0,0,0,0],[9E9,9E9,9E9,9E9,9E9,9E9]];
            P02W26_Approach := [[0,0,0],[1,0,0,0],[0,0,0,0],[9E9,9E9,9E9,9E9,9E9,9E9]];
            P02W26_Retract := [[0,0,0],[1,0,0,0],[0,0,0,0],[9E9,9E9,9E9,9E9,9E9,9E9]];
            P02W26_Trans := [[0,0,0],[1,0,0,0],[0,0,0,0],[9E9,9E9,9E9,9E9,9E9,9E9]];
        ELSEIF slot = 27 THEN
            P02W27_Used := FALSE;
            P02W27_SubType := 0;
            P02W27_ToolSel := 0;
            P02W27_LenMM := 0;
            P02W27_ArcStart := [[0,0,0],[1,0,0,0],[0,0,0,0],[9E9,9E9,9E9,9E9,9E9,9E9]];
            P02W27_ArcEnd := [[0,0,0],[1,0,0,0],[0,0,0,0],[9E9,9E9,9E9,9E9,9E9,9E9]];
            P02W27_Approach := [[0,0,0],[1,0,0,0],[0,0,0,0],[9E9,9E9,9E9,9E9,9E9,9E9]];
            P02W27_Retract := [[0,0,0],[1,0,0,0],[0,0,0,0],[9E9,9E9,9E9,9E9,9E9,9E9]];
            P02W27_Trans := [[0,0,0],[1,0,0,0],[0,0,0,0],[9E9,9E9,9E9,9E9,9E9,9E9]];
        ELSEIF slot = 28 THEN
            P02W28_Used := FALSE;
            P02W28_SubType := 0;
            P02W28_ToolSel := 0;
            P02W28_LenMM := 0;
            P02W28_ArcStart := [[0,0,0],[1,0,0,0],[0,0,0,0],[9E9,9E9,9E9,9E9,9E9,9E9]];
            P02W28_ArcEnd := [[0,0,0],[1,0,0,0],[0,0,0,0],[9E9,9E9,9E9,9E9,9E9,9E9]];
            P02W28_Approach := [[0,0,0],[1,0,0,0],[0,0,0,0],[9E9,9E9,9E9,9E9,9E9,9E9]];
            P02W28_Retract := [[0,0,0],[1,0,0,0],[0,0,0,0],[9E9,9E9,9E9,9E9,9E9,9E9]];
            P02W28_Trans := [[0,0,0],[1,0,0,0],[0,0,0,0],[9E9,9E9,9E9,9E9,9E9,9E9]];
        ELSEIF slot = 29 THEN
            P02W29_Used := FALSE;
            P02W29_SubType := 0;
            P02W29_ToolSel := 0;
            P02W29_LenMM := 0;
            P02W29_ArcStart := [[0,0,0],[1,0,0,0],[0,0,0,0],[9E9,9E9,9E9,9E9,9E9,9E9]];
            P02W29_ArcEnd := [[0,0,0],[1,0,0,0],[0,0,0,0],[9E9,9E9,9E9,9E9,9E9,9E9]];
            P02W29_Approach := [[0,0,0],[1,0,0,0],[0,0,0,0],[9E9,9E9,9E9,9E9,9E9,9E9]];
            P02W29_Retract := [[0,0,0],[1,0,0,0],[0,0,0,0],[9E9,9E9,9E9,9E9,9E9,9E9]];
            P02W29_Trans := [[0,0,0],[1,0,0,0],[0,0,0,0],[9E9,9E9,9E9,9E9,9E9,9E9]];
        ELSEIF slot = 30 THEN
            P02W30_Used := FALSE;
            P02W30_SubType := 0;
            P02W30_ToolSel := 0;
            P02W30_LenMM := 0;
            P02W30_ArcStart := [[0,0,0],[1,0,0,0],[0,0,0,0],[9E9,9E9,9E9,9E9,9E9,9E9]];
            P02W30_ArcEnd := [[0,0,0],[1,0,0,0],[0,0,0,0],[9E9,9E9,9E9,9E9,9E9,9E9]];
            P02W30_Approach := [[0,0,0],[1,0,0,0],[0,0,0,0],[9E9,9E9,9E9,9E9,9E9,9E9]];
            P02W30_Retract := [[0,0,0],[1,0,0,0],[0,0,0,0],[9E9,9E9,9E9,9E9,9E9,9E9]];
            P02W30_Trans := [[0,0,0],[1,0,0,0],[0,0,0,0],[9E9,9E9,9E9,9E9,9E9,9E9]];
        ELSE
            TPWrite "Invalid weld slot.";
        ENDIF
    ENDPROC

    PROC StoreNextFree_P02(num subType, num toolSel, num lenMM,
                       robtarget arcStart, robtarget arcEnd, robtarget approach, robtarget retract, robtarget trans)
        IF NOT P02W01_Used THEN
            StoreSlot_P02 1, subType, toolSel, lenMM, arcStart, arcEnd, approach, retract, trans;
            nWeldsP02 := nWeldsP02 + 1;
            RETURN;
        ELSEIF NOT P02W02_Used THEN
            StoreSlot_P02 2, subType, toolSel, lenMM, arcStart, arcEnd, approach, retract, trans;
            nWeldsP02 := nWeldsP02 + 1;
            RETURN;
        ELSEIF NOT P02W03_Used THEN
            StoreSlot_P02 3, subType, toolSel, lenMM, arcStart, arcEnd, approach, retract, trans;
            nWeldsP02 := nWeldsP02 + 1;
            RETURN;
        ELSEIF NOT P02W04_Used THEN
            StoreSlot_P02 4, subType, toolSel, lenMM, arcStart, arcEnd, approach, retract, trans;
            nWeldsP02 := nWeldsP02 + 1;
            RETURN;
        ELSEIF NOT P02W05_Used THEN
            StoreSlot_P02 5, subType, toolSel, lenMM, arcStart, arcEnd, approach, retract, trans;
            nWeldsP02 := nWeldsP02 + 1;
            RETURN;
        ELSEIF NOT P02W06_Used THEN
            StoreSlot_P02 6, subType, toolSel, lenMM, arcStart, arcEnd, approach, retract, trans;
            nWeldsP02 := nWeldsP02 + 1;
            RETURN;
        ELSEIF NOT P02W07_Used THEN
            StoreSlot_P02 7, subType, toolSel, lenMM, arcStart, arcEnd, approach, retract, trans;
            nWeldsP02 := nWeldsP02 + 1;
            RETURN;
        ELSEIF NOT P02W08_Used THEN
            StoreSlot_P02 8, subType, toolSel, lenMM, arcStart, arcEnd, approach, retract, trans;
            nWeldsP02 := nWeldsP02 + 1;
            RETURN;
        ELSEIF NOT P02W09_Used THEN
            StoreSlot_P02 9, subType, toolSel, lenMM, arcStart, arcEnd, approach, retract, trans;
            nWeldsP02 := nWeldsP02 + 1;
            RETURN;
        ELSEIF NOT P02W10_Used THEN
            StoreSlot_P02 10, subType, toolSel, lenMM, arcStart, arcEnd, approach, retract, trans;
            nWeldsP02 := nWeldsP02 + 1;
            RETURN;
        ELSEIF NOT P02W11_Used THEN
            StoreSlot_P02 11, subType, toolSel, lenMM, arcStart, arcEnd, approach, retract, trans;
            nWeldsP02 := nWeldsP02 + 1;
            RETURN;
        ELSEIF NOT P02W12_Used THEN
            StoreSlot_P02 12, subType, toolSel, lenMM, arcStart, arcEnd, approach, retract, trans;
            nWeldsP02 := nWeldsP02 + 1;
            RETURN;
        ELSEIF NOT P02W13_Used THEN
            StoreSlot_P02 13, subType, toolSel, lenMM, arcStart, arcEnd, approach, retract, trans;
            nWeldsP02 := nWeldsP02 + 1;
            RETURN;
        ELSEIF NOT P02W14_Used THEN
            StoreSlot_P02 14, subType, toolSel, lenMM, arcStart, arcEnd, approach, retract, trans;
            nWeldsP02 := nWeldsP02 + 1;
            RETURN;
        ELSEIF NOT P02W15_Used THEN
            StoreSlot_P02 15, subType, toolSel, lenMM, arcStart, arcEnd, approach, retract, trans;
            nWeldsP02 := nWeldsP02 + 1;
            RETURN;
        ELSEIF NOT P02W16_Used THEN
            StoreSlot_P02 16, subType, toolSel, lenMM, arcStart, arcEnd, approach, retract, trans;
            nWeldsP02 := nWeldsP02 + 1;
            RETURN;
        ELSEIF NOT P02W17_Used THEN
            StoreSlot_P02 17, subType, toolSel, lenMM, arcStart, arcEnd, approach, retract, trans;
            nWeldsP02 := nWeldsP02 + 1;
            RETURN;
        ELSEIF NOT P02W18_Used THEN
            StoreSlot_P02 18, subType, toolSel, lenMM, arcStart, arcEnd, approach, retract, trans;
            nWeldsP02 := nWeldsP02 + 1;
            RETURN;
        ELSEIF NOT P02W19_Used THEN
            StoreSlot_P02 19, subType, toolSel, lenMM, arcStart, arcEnd, approach, retract, trans;
            nWeldsP02 := nWeldsP02 + 1;
            RETURN;
        ELSEIF NOT P02W20_Used THEN
            StoreSlot_P02 20, subType, toolSel, lenMM, arcStart, arcEnd, approach, retract, trans;
            nWeldsP02 := nWeldsP02 + 1;
            RETURN;
        ELSEIF NOT P02W21_Used THEN
            StoreSlot_P02 21, subType, toolSel, lenMM, arcStart, arcEnd, approach, retract, trans;
            nWeldsP02 := nWeldsP02 + 1;
            RETURN;
        ELSEIF NOT P02W22_Used THEN
            StoreSlot_P02 22, subType, toolSel, lenMM, arcStart, arcEnd, approach, retract, trans;
            nWeldsP02 := nWeldsP02 + 1;
            RETURN;
        ELSEIF NOT P02W23_Used THEN
            StoreSlot_P02 23, subType, toolSel, lenMM, arcStart, arcEnd, approach, retract, trans;
            nWeldsP02 := nWeldsP02 + 1;
            RETURN;
        ELSEIF NOT P02W24_Used THEN
            StoreSlot_P02 24, subType, toolSel, lenMM, arcStart, arcEnd, approach, retract, trans;
            nWeldsP02 := nWeldsP02 + 1;
            RETURN;
        ELSEIF NOT P02W25_Used THEN
            StoreSlot_P02 25, subType, toolSel, lenMM, arcStart, arcEnd, approach, retract, trans;
            nWeldsP02 := nWeldsP02 + 1;
            RETURN;
        ELSEIF NOT P02W26_Used THEN
            StoreSlot_P02 26, subType, toolSel, lenMM, arcStart, arcEnd, approach, retract, trans;
            nWeldsP02 := nWeldsP02 + 1;
            RETURN;
        ELSEIF NOT P02W27_Used THEN
            StoreSlot_P02 27, subType, toolSel, lenMM, arcStart, arcEnd, approach, retract, trans;
            nWeldsP02 := nWeldsP02 + 1;
            RETURN;
        ELSEIF NOT P02W28_Used THEN
            StoreSlot_P02 28, subType, toolSel, lenMM, arcStart, arcEnd, approach, retract, trans;
            nWeldsP02 := nWeldsP02 + 1;
            RETURN;
        ELSEIF NOT P02W29_Used THEN
            StoreSlot_P02 29, subType, toolSel, lenMM, arcStart, arcEnd, approach, retract, trans;
            nWeldsP02 := nWeldsP02 + 1;
            RETURN;
        ELSEIF NOT P02W30_Used THEN
            StoreSlot_P02 30, subType, toolSel, lenMM, arcStart, arcEnd, approach, retract, trans;
            nWeldsP02 := nWeldsP02 + 1;
            RETURN;
        ELSE
            TPWrite "No free weld slots available.";
        ENDIF
    ENDPROC

    PROC StoreSlot_P03(num slot, num subType, num toolSel, num lenMM,
                       robtarget arcStart, robtarget arcEnd, robtarget approach, robtarget retract, robtarget trans)
        IF slot = 1 THEN
            P03W01_SubType := subType;
            P03W01_ToolSel := toolSel;
            P03W01_LenMM := lenMM;
            P03W01_ArcStart := arcStart;
            P03W01_ArcEnd := arcEnd;
            P03W01_Approach := approach;
            P03W01_Retract := retract;
            P03W01_Trans := trans;
            P03W01_Used := TRUE;
        ELSEIF slot = 2 THEN
            P03W02_SubType := subType;
            P03W02_ToolSel := toolSel;
            P03W02_LenMM := lenMM;
            P03W02_ArcStart := arcStart;
            P03W02_ArcEnd := arcEnd;
            P03W02_Approach := approach;
            P03W02_Retract := retract;
            P03W02_Trans := trans;
            P03W02_Used := TRUE;
        ELSEIF slot = 3 THEN
            P03W03_SubType := subType;
            P03W03_ToolSel := toolSel;
            P03W03_LenMM := lenMM;
            P03W03_ArcStart := arcStart;
            P03W03_ArcEnd := arcEnd;
            P03W03_Approach := approach;
            P03W03_Retract := retract;
            P03W03_Trans := trans;
            P03W03_Used := TRUE;
        ELSEIF slot = 4 THEN
            P03W04_SubType := subType;
            P03W04_ToolSel := toolSel;
            P03W04_LenMM := lenMM;
            P03W04_ArcStart := arcStart;
            P03W04_ArcEnd := arcEnd;
            P03W04_Approach := approach;
            P03W04_Retract := retract;
            P03W04_Trans := trans;
            P03W04_Used := TRUE;
        ELSEIF slot = 5 THEN
            P03W05_SubType := subType;
            P03W05_ToolSel := toolSel;
            P03W05_LenMM := lenMM;
            P03W05_ArcStart := arcStart;
            P03W05_ArcEnd := arcEnd;
            P03W05_Approach := approach;
            P03W05_Retract := retract;
            P03W05_Trans := trans;
            P03W05_Used := TRUE;
        ELSEIF slot = 6 THEN
            P03W06_SubType := subType;
            P03W06_ToolSel := toolSel;
            P03W06_LenMM := lenMM;
            P03W06_ArcStart := arcStart;
            P03W06_ArcEnd := arcEnd;
            P03W06_Approach := approach;
            P03W06_Retract := retract;
            P03W06_Trans := trans;
            P03W06_Used := TRUE;
        ELSEIF slot = 7 THEN
            P03W07_SubType := subType;
            P03W07_ToolSel := toolSel;
            P03W07_LenMM := lenMM;
            P03W07_ArcStart := arcStart;
            P03W07_ArcEnd := arcEnd;
            P03W07_Approach := approach;
            P03W07_Retract := retract;
            P03W07_Trans := trans;
            P03W07_Used := TRUE;
        ELSEIF slot = 8 THEN
            P03W08_SubType := subType;
            P03W08_ToolSel := toolSel;
            P03W08_LenMM := lenMM;
            P03W08_ArcStart := arcStart;
            P03W08_ArcEnd := arcEnd;
            P03W08_Approach := approach;
            P03W08_Retract := retract;
            P03W08_Trans := trans;
            P03W08_Used := TRUE;
        ELSEIF slot = 9 THEN
            P03W09_SubType := subType;
            P03W09_ToolSel := toolSel;
            P03W09_LenMM := lenMM;
            P03W09_ArcStart := arcStart;
            P03W09_ArcEnd := arcEnd;
            P03W09_Approach := approach;
            P03W09_Retract := retract;
            P03W09_Trans := trans;
            P03W09_Used := TRUE;
        ELSEIF slot = 10 THEN
            P03W10_SubType := subType;
            P03W10_ToolSel := toolSel;
            P03W10_LenMM := lenMM;
            P03W10_ArcStart := arcStart;
            P03W10_ArcEnd := arcEnd;
            P03W10_Approach := approach;
            P03W10_Retract := retract;
            P03W10_Trans := trans;
            P03W10_Used := TRUE;
        ELSEIF slot = 11 THEN
            P03W11_SubType := subType;
            P03W11_ToolSel := toolSel;
            P03W11_LenMM := lenMM;
            P03W11_ArcStart := arcStart;
            P03W11_ArcEnd := arcEnd;
            P03W11_Approach := approach;
            P03W11_Retract := retract;
            P03W11_Trans := trans;
            P03W11_Used := TRUE;
        ELSEIF slot = 12 THEN
            P03W12_SubType := subType;
            P03W12_ToolSel := toolSel;
            P03W12_LenMM := lenMM;
            P03W12_ArcStart := arcStart;
            P03W12_ArcEnd := arcEnd;
            P03W12_Approach := approach;
            P03W12_Retract := retract;
            P03W12_Trans := trans;
            P03W12_Used := TRUE;
        ELSEIF slot = 13 THEN
            P03W13_SubType := subType;
            P03W13_ToolSel := toolSel;
            P03W13_LenMM := lenMM;
            P03W13_ArcStart := arcStart;
            P03W13_ArcEnd := arcEnd;
            P03W13_Approach := approach;
            P03W13_Retract := retract;
            P03W13_Trans := trans;
            P03W13_Used := TRUE;
        ELSEIF slot = 14 THEN
            P03W14_SubType := subType;
            P03W14_ToolSel := toolSel;
            P03W14_LenMM := lenMM;
            P03W14_ArcStart := arcStart;
            P03W14_ArcEnd := arcEnd;
            P03W14_Approach := approach;
            P03W14_Retract := retract;
            P03W14_Trans := trans;
            P03W14_Used := TRUE;
        ELSEIF slot = 15 THEN
            P03W15_SubType := subType;
            P03W15_ToolSel := toolSel;
            P03W15_LenMM := lenMM;
            P03W15_ArcStart := arcStart;
            P03W15_ArcEnd := arcEnd;
            P03W15_Approach := approach;
            P03W15_Retract := retract;
            P03W15_Trans := trans;
            P03W15_Used := TRUE;
        ELSEIF slot = 16 THEN
            P03W16_SubType := subType;
            P03W16_ToolSel := toolSel;
            P03W16_LenMM := lenMM;
            P03W16_ArcStart := arcStart;
            P03W16_ArcEnd := arcEnd;
            P03W16_Approach := approach;
            P03W16_Retract := retract;
            P03W16_Trans := trans;
            P03W16_Used := TRUE;
        ELSEIF slot = 17 THEN
            P03W17_SubType := subType;
            P03W17_ToolSel := toolSel;
            P03W17_LenMM := lenMM;
            P03W17_ArcStart := arcStart;
            P03W17_ArcEnd := arcEnd;
            P03W17_Approach := approach;
            P03W17_Retract := retract;
            P03W17_Trans := trans;
            P03W17_Used := TRUE;
        ELSEIF slot = 18 THEN
            P03W18_SubType := subType;
            P03W18_ToolSel := toolSel;
            P03W18_LenMM := lenMM;
            P03W18_ArcStart := arcStart;
            P03W18_ArcEnd := arcEnd;
            P03W18_Approach := approach;
            P03W18_Retract := retract;
            P03W18_Trans := trans;
            P03W18_Used := TRUE;
        ELSEIF slot = 19 THEN
            P03W19_SubType := subType;
            P03W19_ToolSel := toolSel;
            P03W19_LenMM := lenMM;
            P03W19_ArcStart := arcStart;
            P03W19_ArcEnd := arcEnd;
            P03W19_Approach := approach;
            P03W19_Retract := retract;
            P03W19_Trans := trans;
            P03W19_Used := TRUE;
        ELSEIF slot = 20 THEN
            P03W20_SubType := subType;
            P03W20_ToolSel := toolSel;
            P03W20_LenMM := lenMM;
            P03W20_ArcStart := arcStart;
            P03W20_ArcEnd := arcEnd;
            P03W20_Approach := approach;
            P03W20_Retract := retract;
            P03W20_Trans := trans;
            P03W20_Used := TRUE;
        ELSEIF slot = 21 THEN
            P03W21_SubType := subType;
            P03W21_ToolSel := toolSel;
            P03W21_LenMM := lenMM;
            P03W21_ArcStart := arcStart;
            P03W21_ArcEnd := arcEnd;
            P03W21_Approach := approach;
            P03W21_Retract := retract;
            P03W21_Trans := trans;
            P03W21_Used := TRUE;
        ELSEIF slot = 22 THEN
            P03W22_SubType := subType;
            P03W22_ToolSel := toolSel;
            P03W22_LenMM := lenMM;
            P03W22_ArcStart := arcStart;
            P03W22_ArcEnd := arcEnd;
            P03W22_Approach := approach;
            P03W22_Retract := retract;
            P03W22_Trans := trans;
            P03W22_Used := TRUE;
        ELSEIF slot = 23 THEN
            P03W23_SubType := subType;
            P03W23_ToolSel := toolSel;
            P03W23_LenMM := lenMM;
            P03W23_ArcStart := arcStart;
            P03W23_ArcEnd := arcEnd;
            P03W23_Approach := approach;
            P03W23_Retract := retract;
            P03W23_Trans := trans;
            P03W23_Used := TRUE;
        ELSEIF slot = 24 THEN
            P03W24_SubType := subType;
            P03W24_ToolSel := toolSel;
            P03W24_LenMM := lenMM;
            P03W24_ArcStart := arcStart;
            P03W24_ArcEnd := arcEnd;
            P03W24_Approach := approach;
            P03W24_Retract := retract;
            P03W24_Trans := trans;
            P03W24_Used := TRUE;
        ELSEIF slot = 25 THEN
            P03W25_SubType := subType;
            P03W25_ToolSel := toolSel;
            P03W25_LenMM := lenMM;
            P03W25_ArcStart := arcStart;
            P03W25_ArcEnd := arcEnd;
            P03W25_Approach := approach;
            P03W25_Retract := retract;
            P03W25_Trans := trans;
            P03W25_Used := TRUE;
        ELSEIF slot = 26 THEN
            P03W26_SubType := subType;
            P03W26_ToolSel := toolSel;
            P03W26_LenMM := lenMM;
            P03W26_ArcStart := arcStart;
            P03W26_ArcEnd := arcEnd;
            P03W26_Approach := approach;
            P03W26_Retract := retract;
            P03W26_Trans := trans;
            P03W26_Used := TRUE;
        ELSEIF slot = 27 THEN
            P03W27_SubType := subType;
            P03W27_ToolSel := toolSel;
            P03W27_LenMM := lenMM;
            P03W27_ArcStart := arcStart;
            P03W27_ArcEnd := arcEnd;
            P03W27_Approach := approach;
            P03W27_Retract := retract;
            P03W27_Trans := trans;
            P03W27_Used := TRUE;
        ELSEIF slot = 28 THEN
            P03W28_SubType := subType;
            P03W28_ToolSel := toolSel;
            P03W28_LenMM := lenMM;
            P03W28_ArcStart := arcStart;
            P03W28_ArcEnd := arcEnd;
            P03W28_Approach := approach;
            P03W28_Retract := retract;
            P03W28_Trans := trans;
            P03W28_Used := TRUE;
        ELSEIF slot = 29 THEN
            P03W29_SubType := subType;
            P03W29_ToolSel := toolSel;
            P03W29_LenMM := lenMM;
            P03W29_ArcStart := arcStart;
            P03W29_ArcEnd := arcEnd;
            P03W29_Approach := approach;
            P03W29_Retract := retract;
            P03W29_Trans := trans;
            P03W29_Used := TRUE;
        ELSEIF slot = 30 THEN
            P03W30_SubType := subType;
            P03W30_ToolSel := toolSel;
            P03W30_LenMM := lenMM;
            P03W30_ArcStart := arcStart;
            P03W30_ArcEnd := arcEnd;
            P03W30_Approach := approach;
            P03W30_Retract := retract;
            P03W30_Trans := trans;
            P03W30_Used := TRUE;
        ELSE
            TPWrite "Invalid weld slot.";
        ENDIF
    ENDPROC

    PROC LoadSlot_P03(num slot, VAR bool used, VAR num subType, VAR num toolSel, VAR num lenMM,
                       VAR robtarget arcStart, VAR robtarget arcEnd, VAR robtarget approach, VAR robtarget retract, VAR robtarget trans)
        IF slot = 1 THEN
            used := P03W01_Used;
            subType := P03W01_SubType;
            toolSel := P03W01_ToolSel;
            lenMM := P03W01_LenMM;
            arcStart := P03W01_ArcStart;
            arcEnd := P03W01_ArcEnd;
            approach := P03W01_Approach;
            retract := P03W01_Retract;
            trans := P03W01_Trans;
        ELSEIF slot = 2 THEN
            used := P03W02_Used;
            subType := P03W02_SubType;
            toolSel := P03W02_ToolSel;
            lenMM := P03W02_LenMM;
            arcStart := P03W02_ArcStart;
            arcEnd := P03W02_ArcEnd;
            approach := P03W02_Approach;
            retract := P03W02_Retract;
            trans := P03W02_Trans;
        ELSEIF slot = 3 THEN
            used := P03W03_Used;
            subType := P03W03_SubType;
            toolSel := P03W03_ToolSel;
            lenMM := P03W03_LenMM;
            arcStart := P03W03_ArcStart;
            arcEnd := P03W03_ArcEnd;
            approach := P03W03_Approach;
            retract := P03W03_Retract;
            trans := P03W03_Trans;
        ELSEIF slot = 4 THEN
            used := P03W04_Used;
            subType := P03W04_SubType;
            toolSel := P03W04_ToolSel;
            lenMM := P03W04_LenMM;
            arcStart := P03W04_ArcStart;
            arcEnd := P03W04_ArcEnd;
            approach := P03W04_Approach;
            retract := P03W04_Retract;
            trans := P03W04_Trans;
        ELSEIF slot = 5 THEN
            used := P03W05_Used;
            subType := P03W05_SubType;
            toolSel := P03W05_ToolSel;
            lenMM := P03W05_LenMM;
            arcStart := P03W05_ArcStart;
            arcEnd := P03W05_ArcEnd;
            approach := P03W05_Approach;
            retract := P03W05_Retract;
            trans := P03W05_Trans;
        ELSEIF slot = 6 THEN
            used := P03W06_Used;
            subType := P03W06_SubType;
            toolSel := P03W06_ToolSel;
            lenMM := P03W06_LenMM;
            arcStart := P03W06_ArcStart;
            arcEnd := P03W06_ArcEnd;
            approach := P03W06_Approach;
            retract := P03W06_Retract;
            trans := P03W06_Trans;
        ELSEIF slot = 7 THEN
            used := P03W07_Used;
            subType := P03W07_SubType;
            toolSel := P03W07_ToolSel;
            lenMM := P03W07_LenMM;
            arcStart := P03W07_ArcStart;
            arcEnd := P03W07_ArcEnd;
            approach := P03W07_Approach;
            retract := P03W07_Retract;
            trans := P03W07_Trans;
        ELSEIF slot = 8 THEN
            used := P03W08_Used;
            subType := P03W08_SubType;
            toolSel := P03W08_ToolSel;
            lenMM := P03W08_LenMM;
            arcStart := P03W08_ArcStart;
            arcEnd := P03W08_ArcEnd;
            approach := P03W08_Approach;
            retract := P03W08_Retract;
            trans := P03W08_Trans;
        ELSEIF slot = 9 THEN
            used := P03W09_Used;
            subType := P03W09_SubType;
            toolSel := P03W09_ToolSel;
            lenMM := P03W09_LenMM;
            arcStart := P03W09_ArcStart;
            arcEnd := P03W09_ArcEnd;
            approach := P03W09_Approach;
            retract := P03W09_Retract;
            trans := P03W09_Trans;
        ELSEIF slot = 10 THEN
            used := P03W10_Used;
            subType := P03W10_SubType;
            toolSel := P03W10_ToolSel;
            lenMM := P03W10_LenMM;
            arcStart := P03W10_ArcStart;
            arcEnd := P03W10_ArcEnd;
            approach := P03W10_Approach;
            retract := P03W10_Retract;
            trans := P03W10_Trans;
        ELSEIF slot = 11 THEN
            used := P03W11_Used;
            subType := P03W11_SubType;
            toolSel := P03W11_ToolSel;
            lenMM := P03W11_LenMM;
            arcStart := P03W11_ArcStart;
            arcEnd := P03W11_ArcEnd;
            approach := P03W11_Approach;
            retract := P03W11_Retract;
            trans := P03W11_Trans;
        ELSEIF slot = 12 THEN
            used := P03W12_Used;
            subType := P03W12_SubType;
            toolSel := P03W12_ToolSel;
            lenMM := P03W12_LenMM;
            arcStart := P03W12_ArcStart;
            arcEnd := P03W12_ArcEnd;
            approach := P03W12_Approach;
            retract := P03W12_Retract;
            trans := P03W12_Trans;
        ELSEIF slot = 13 THEN
            used := P03W13_Used;
            subType := P03W13_SubType;
            toolSel := P03W13_ToolSel;
            lenMM := P03W13_LenMM;
            arcStart := P03W13_ArcStart;
            arcEnd := P03W13_ArcEnd;
            approach := P03W13_Approach;
            retract := P03W13_Retract;
            trans := P03W13_Trans;
        ELSEIF slot = 14 THEN
            used := P03W14_Used;
            subType := P03W14_SubType;
            toolSel := P03W14_ToolSel;
            lenMM := P03W14_LenMM;
            arcStart := P03W14_ArcStart;
            arcEnd := P03W14_ArcEnd;
            approach := P03W14_Approach;
            retract := P03W14_Retract;
            trans := P03W14_Trans;
        ELSEIF slot = 15 THEN
            used := P03W15_Used;
            subType := P03W15_SubType;
            toolSel := P03W15_ToolSel;
            lenMM := P03W15_LenMM;
            arcStart := P03W15_ArcStart;
            arcEnd := P03W15_ArcEnd;
            approach := P03W15_Approach;
            retract := P03W15_Retract;
            trans := P03W15_Trans;
        ELSEIF slot = 16 THEN
            used := P03W16_Used;
            subType := P03W16_SubType;
            toolSel := P03W16_ToolSel;
            lenMM := P03W16_LenMM;
            arcStart := P03W16_ArcStart;
            arcEnd := P03W16_ArcEnd;
            approach := P03W16_Approach;
            retract := P03W16_Retract;
            trans := P03W16_Trans;
        ELSEIF slot = 17 THEN
            used := P03W17_Used;
            subType := P03W17_SubType;
            toolSel := P03W17_ToolSel;
            lenMM := P03W17_LenMM;
            arcStart := P03W17_ArcStart;
            arcEnd := P03W17_ArcEnd;
            approach := P03W17_Approach;
            retract := P03W17_Retract;
            trans := P03W17_Trans;
        ELSEIF slot = 18 THEN
            used := P03W18_Used;
            subType := P03W18_SubType;
            toolSel := P03W18_ToolSel;
            lenMM := P03W18_LenMM;
            arcStart := P03W18_ArcStart;
            arcEnd := P03W18_ArcEnd;
            approach := P03W18_Approach;
            retract := P03W18_Retract;
            trans := P03W18_Trans;
        ELSEIF slot = 19 THEN
            used := P03W19_Used;
            subType := P03W19_SubType;
            toolSel := P03W19_ToolSel;
            lenMM := P03W19_LenMM;
            arcStart := P03W19_ArcStart;
            arcEnd := P03W19_ArcEnd;
            approach := P03W19_Approach;
            retract := P03W19_Retract;
            trans := P03W19_Trans;
        ELSEIF slot = 20 THEN
            used := P03W20_Used;
            subType := P03W20_SubType;
            toolSel := P03W20_ToolSel;
            lenMM := P03W20_LenMM;
            arcStart := P03W20_ArcStart;
            arcEnd := P03W20_ArcEnd;
            approach := P03W20_Approach;
            retract := P03W20_Retract;
            trans := P03W20_Trans;
        ELSEIF slot = 21 THEN
            used := P03W21_Used;
            subType := P03W21_SubType;
            toolSel := P03W21_ToolSel;
            lenMM := P03W21_LenMM;
            arcStart := P03W21_ArcStart;
            arcEnd := P03W21_ArcEnd;
            approach := P03W21_Approach;
            retract := P03W21_Retract;
            trans := P03W21_Trans;
        ELSEIF slot = 22 THEN
            used := P03W22_Used;
            subType := P03W22_SubType;
            toolSel := P03W22_ToolSel;
            lenMM := P03W22_LenMM;
            arcStart := P03W22_ArcStart;
            arcEnd := P03W22_ArcEnd;
            approach := P03W22_Approach;
            retract := P03W22_Retract;
            trans := P03W22_Trans;
        ELSEIF slot = 23 THEN
            used := P03W23_Used;
            subType := P03W23_SubType;
            toolSel := P03W23_ToolSel;
            lenMM := P03W23_LenMM;
            arcStart := P03W23_ArcStart;
            arcEnd := P03W23_ArcEnd;
            approach := P03W23_Approach;
            retract := P03W23_Retract;
            trans := P03W23_Trans;
        ELSEIF slot = 24 THEN
            used := P03W24_Used;
            subType := P03W24_SubType;
            toolSel := P03W24_ToolSel;
            lenMM := P03W24_LenMM;
            arcStart := P03W24_ArcStart;
            arcEnd := P03W24_ArcEnd;
            approach := P03W24_Approach;
            retract := P03W24_Retract;
            trans := P03W24_Trans;
        ELSEIF slot = 25 THEN
            used := P03W25_Used;
            subType := P03W25_SubType;
            toolSel := P03W25_ToolSel;
            lenMM := P03W25_LenMM;
            arcStart := P03W25_ArcStart;
            arcEnd := P03W25_ArcEnd;
            approach := P03W25_Approach;
            retract := P03W25_Retract;
            trans := P03W25_Trans;
        ELSEIF slot = 26 THEN
            used := P03W26_Used;
            subType := P03W26_SubType;
            toolSel := P03W26_ToolSel;
            lenMM := P03W26_LenMM;
            arcStart := P03W26_ArcStart;
            arcEnd := P03W26_ArcEnd;
            approach := P03W26_Approach;
            retract := P03W26_Retract;
            trans := P03W26_Trans;
        ELSEIF slot = 27 THEN
            used := P03W27_Used;
            subType := P03W27_SubType;
            toolSel := P03W27_ToolSel;
            lenMM := P03W27_LenMM;
            arcStart := P03W27_ArcStart;
            arcEnd := P03W27_ArcEnd;
            approach := P03W27_Approach;
            retract := P03W27_Retract;
            trans := P03W27_Trans;
        ELSEIF slot = 28 THEN
            used := P03W28_Used;
            subType := P03W28_SubType;
            toolSel := P03W28_ToolSel;
            lenMM := P03W28_LenMM;
            arcStart := P03W28_ArcStart;
            arcEnd := P03W28_ArcEnd;
            approach := P03W28_Approach;
            retract := P03W28_Retract;
            trans := P03W28_Trans;
        ELSEIF slot = 29 THEN
            used := P03W29_Used;
            subType := P03W29_SubType;
            toolSel := P03W29_ToolSel;
            lenMM := P03W29_LenMM;
            arcStart := P03W29_ArcStart;
            arcEnd := P03W29_ArcEnd;
            approach := P03W29_Approach;
            retract := P03W29_Retract;
            trans := P03W29_Trans;
        ELSEIF slot = 30 THEN
            used := P03W30_Used;
            subType := P03W30_SubType;
            toolSel := P03W30_ToolSel;
            lenMM := P03W30_LenMM;
            arcStart := P03W30_ArcStart;
            arcEnd := P03W30_ArcEnd;
            approach := P03W30_Approach;
            retract := P03W30_Retract;
            trans := P03W30_Trans;
        ELSE
            used := FALSE;
        ENDIF
    ENDPROC

    PROC ClearSlot_P03(num slot)
        IF slot = 1 THEN
            P03W01_Used := FALSE;
            P03W01_SubType := 0;
            P03W01_ToolSel := 0;
            P03W01_LenMM := 0;
            P03W01_ArcStart := [[0,0,0],[1,0,0,0],[0,0,0,0],[9E9,9E9,9E9,9E9,9E9,9E9]];
            P03W01_ArcEnd := [[0,0,0],[1,0,0,0],[0,0,0,0],[9E9,9E9,9E9,9E9,9E9,9E9]];
            P03W01_Approach := [[0,0,0],[1,0,0,0],[0,0,0,0],[9E9,9E9,9E9,9E9,9E9,9E9]];
            P03W01_Retract := [[0,0,0],[1,0,0,0],[0,0,0,0],[9E9,9E9,9E9,9E9,9E9,9E9]];
            P03W01_Trans := [[0,0,0],[1,0,0,0],[0,0,0,0],[9E9,9E9,9E9,9E9,9E9,9E9]];
        ELSEIF slot = 2 THEN
            P03W02_Used := FALSE;
            P03W02_SubType := 0;
            P03W02_ToolSel := 0;
            P03W02_LenMM := 0;
            P03W02_ArcStart := [[0,0,0],[1,0,0,0],[0,0,0,0],[9E9,9E9,9E9,9E9,9E9,9E9]];
            P03W02_ArcEnd := [[0,0,0],[1,0,0,0],[0,0,0,0],[9E9,9E9,9E9,9E9,9E9,9E9]];
            P03W02_Approach := [[0,0,0],[1,0,0,0],[0,0,0,0],[9E9,9E9,9E9,9E9,9E9,9E9]];
            P03W02_Retract := [[0,0,0],[1,0,0,0],[0,0,0,0],[9E9,9E9,9E9,9E9,9E9,9E9]];
            P03W02_Trans := [[0,0,0],[1,0,0,0],[0,0,0,0],[9E9,9E9,9E9,9E9,9E9,9E9]];
        ELSEIF slot = 3 THEN
            P03W03_Used := FALSE;
            P03W03_SubType := 0;
            P03W03_ToolSel := 0;
            P03W03_LenMM := 0;
            P03W03_ArcStart := [[0,0,0],[1,0,0,0],[0,0,0,0],[9E9,9E9,9E9,9E9,9E9,9E9]];
            P03W03_ArcEnd := [[0,0,0],[1,0,0,0],[0,0,0,0],[9E9,9E9,9E9,9E9,9E9,9E9]];
            P03W03_Approach := [[0,0,0],[1,0,0,0],[0,0,0,0],[9E9,9E9,9E9,9E9,9E9,9E9]];
            P03W03_Retract := [[0,0,0],[1,0,0,0],[0,0,0,0],[9E9,9E9,9E9,9E9,9E9,9E9]];
            P03W03_Trans := [[0,0,0],[1,0,0,0],[0,0,0,0],[9E9,9E9,9E9,9E9,9E9,9E9]];
        ELSEIF slot = 4 THEN
            P03W04_Used := FALSE;
            P03W04_SubType := 0;
            P03W04_ToolSel := 0;
            P03W04_LenMM := 0;
            P03W04_ArcStart := [[0,0,0],[1,0,0,0],[0,0,0,0],[9E9,9E9,9E9,9E9,9E9,9E9]];
            P03W04_ArcEnd := [[0,0,0],[1,0,0,0],[0,0,0,0],[9E9,9E9,9E9,9E9,9E9,9E9]];
            P03W04_Approach := [[0,0,0],[1,0,0,0],[0,0,0,0],[9E9,9E9,9E9,9E9,9E9,9E9]];
            P03W04_Retract := [[0,0,0],[1,0,0,0],[0,0,0,0],[9E9,9E9,9E9,9E9,9E9,9E9]];
            P03W04_Trans := [[0,0,0],[1,0,0,0],[0,0,0,0],[9E9,9E9,9E9,9E9,9E9,9E9]];
        ELSEIF slot = 5 THEN
            P03W05_Used := FALSE;
            P03W05_SubType := 0;
            P03W05_ToolSel := 0;
            P03W05_LenMM := 0;
            P03W05_ArcStart := [[0,0,0],[1,0,0,0],[0,0,0,0],[9E9,9E9,9E9,9E9,9E9,9E9]];
            P03W05_ArcEnd := [[0,0,0],[1,0,0,0],[0,0,0,0],[9E9,9E9,9E9,9E9,9E9,9E9]];
            P03W05_Approach := [[0,0,0],[1,0,0,0],[0,0,0,0],[9E9,9E9,9E9,9E9,9E9,9E9]];
            P03W05_Retract := [[0,0,0],[1,0,0,0],[0,0,0,0],[9E9,9E9,9E9,9E9,9E9,9E9]];
            P03W05_Trans := [[0,0,0],[1,0,0,0],[0,0,0,0],[9E9,9E9,9E9,9E9,9E9,9E9]];
        ELSEIF slot = 6 THEN
            P03W06_Used := FALSE;
            P03W06_SubType := 0;
            P03W06_ToolSel := 0;
            P03W06_LenMM := 0;
            P03W06_ArcStart := [[0,0,0],[1,0,0,0],[0,0,0,0],[9E9,9E9,9E9,9E9,9E9,9E9]];
            P03W06_ArcEnd := [[0,0,0],[1,0,0,0],[0,0,0,0],[9E9,9E9,9E9,9E9,9E9,9E9]];
            P03W06_Approach := [[0,0,0],[1,0,0,0],[0,0,0,0],[9E9,9E9,9E9,9E9,9E9,9E9]];
            P03W06_Retract := [[0,0,0],[1,0,0,0],[0,0,0,0],[9E9,9E9,9E9,9E9,9E9,9E9]];
            P03W06_Trans := [[0,0,0],[1,0,0,0],[0,0,0,0],[9E9,9E9,9E9,9E9,9E9,9E9]];
        ELSEIF slot = 7 THEN
            P03W07_Used := FALSE;
            P03W07_SubType := 0;
            P03W07_ToolSel := 0;
            P03W07_LenMM := 0;
            P03W07_ArcStart := [[0,0,0],[1,0,0,0],[0,0,0,0],[9E9,9E9,9E9,9E9,9E9,9E9]];
            P03W07_ArcEnd := [[0,0,0],[1,0,0,0],[0,0,0,0],[9E9,9E9,9E9,9E9,9E9,9E9]];
            P03W07_Approach := [[0,0,0],[1,0,0,0],[0,0,0,0],[9E9,9E9,9E9,9E9,9E9,9E9]];
            P03W07_Retract := [[0,0,0],[1,0,0,0],[0,0,0,0],[9E9,9E9,9E9,9E9,9E9,9E9]];
            P03W07_Trans := [[0,0,0],[1,0,0,0],[0,0,0,0],[9E9,9E9,9E9,9E9,9E9,9E9]];
        ELSEIF slot = 8 THEN
            P03W08_Used := FALSE;
            P03W08_SubType := 0;
            P03W08_ToolSel := 0;
            P03W08_LenMM := 0;
            P03W08_ArcStart := [[0,0,0],[1,0,0,0],[0,0,0,0],[9E9,9E9,9E9,9E9,9E9,9E9]];
            P03W08_ArcEnd := [[0,0,0],[1,0,0,0],[0,0,0,0],[9E9,9E9,9E9,9E9,9E9,9E9]];
            P03W08_Approach := [[0,0,0],[1,0,0,0],[0,0,0,0],[9E9,9E9,9E9,9E9,9E9,9E9]];
            P03W08_Retract := [[0,0,0],[1,0,0,0],[0,0,0,0],[9E9,9E9,9E9,9E9,9E9,9E9]];
            P03W08_Trans := [[0,0,0],[1,0,0,0],[0,0,0,0],[9E9,9E9,9E9,9E9,9E9,9E9]];
        ELSEIF slot = 9 THEN
            P03W09_Used := FALSE;
            P03W09_SubType := 0;
            P03W09_ToolSel := 0;
            P03W09_LenMM := 0;
            P03W09_ArcStart := [[0,0,0],[1,0,0,0],[0,0,0,0],[9E9,9E9,9E9,9E9,9E9,9E9]];
            P03W09_ArcEnd := [[0,0,0],[1,0,0,0],[0,0,0,0],[9E9,9E9,9E9,9E9,9E9,9E9]];
            P03W09_Approach := [[0,0,0],[1,0,0,0],[0,0,0,0],[9E9,9E9,9E9,9E9,9E9,9E9]];
            P03W09_Retract := [[0,0,0],[1,0,0,0],[0,0,0,0],[9E9,9E9,9E9,9E9,9E9,9E9]];
            P03W09_Trans := [[0,0,0],[1,0,0,0],[0,0,0,0],[9E9,9E9,9E9,9E9,9E9,9E9]];
        ELSEIF slot = 10 THEN
            P03W10_Used := FALSE;
            P03W10_SubType := 0;
            P03W10_ToolSel := 0;
            P03W10_LenMM := 0;
            P03W10_ArcStart := [[0,0,0],[1,0,0,0],[0,0,0,0],[9E9,9E9,9E9,9E9,9E9,9E9]];
            P03W10_ArcEnd := [[0,0,0],[1,0,0,0],[0,0,0,0],[9E9,9E9,9E9,9E9,9E9,9E9]];
            P03W10_Approach := [[0,0,0],[1,0,0,0],[0,0,0,0],[9E9,9E9,9E9,9E9,9E9,9E9]];
            P03W10_Retract := [[0,0,0],[1,0,0,0],[0,0,0,0],[9E9,9E9,9E9,9E9,9E9,9E9]];
            P03W10_Trans := [[0,0,0],[1,0,0,0],[0,0,0,0],[9E9,9E9,9E9,9E9,9E9,9E9]];
        ELSEIF slot = 11 THEN
            P03W11_Used := FALSE;
            P03W11_SubType := 0;
            P03W11_ToolSel := 0;
            P03W11_LenMM := 0;
            P03W11_ArcStart := [[0,0,0],[1,0,0,0],[0,0,0,0],[9E9,9E9,9E9,9E9,9E9,9E9]];
            P03W11_ArcEnd := [[0,0,0],[1,0,0,0],[0,0,0,0],[9E9,9E9,9E9,9E9,9E9,9E9]];
            P03W11_Approach := [[0,0,0],[1,0,0,0],[0,0,0,0],[9E9,9E9,9E9,9E9,9E9,9E9]];
            P03W11_Retract := [[0,0,0],[1,0,0,0],[0,0,0,0],[9E9,9E9,9E9,9E9,9E9,9E9]];
            P03W11_Trans := [[0,0,0],[1,0,0,0],[0,0,0,0],[9E9,9E9,9E9,9E9,9E9,9E9]];
        ELSEIF slot = 12 THEN
            P03W12_Used := FALSE;
            P03W12_SubType := 0;
            P03W12_ToolSel := 0;
            P03W12_LenMM := 0;
            P03W12_ArcStart := [[0,0,0],[1,0,0,0],[0,0,0,0],[9E9,9E9,9E9,9E9,9E9,9E9]];
            P03W12_ArcEnd := [[0,0,0],[1,0,0,0],[0,0,0,0],[9E9,9E9,9E9,9E9,9E9,9E9]];
            P03W12_Approach := [[0,0,0],[1,0,0,0],[0,0,0,0],[9E9,9E9,9E9,9E9,9E9,9E9]];
            P03W12_Retract := [[0,0,0],[1,0,0,0],[0,0,0,0],[9E9,9E9,9E9,9E9,9E9,9E9]];
            P03W12_Trans := [[0,0,0],[1,0,0,0],[0,0,0,0],[9E9,9E9,9E9,9E9,9E9,9E9]];
        ELSEIF slot = 13 THEN
            P03W13_Used := FALSE;
            P03W13_SubType := 0;
            P03W13_ToolSel := 0;
            P03W13_LenMM := 0;
            P03W13_ArcStart := [[0,0,0],[1,0,0,0],[0,0,0,0],[9E9,9E9,9E9,9E9,9E9,9E9]];
            P03W13_ArcEnd := [[0,0,0],[1,0,0,0],[0,0,0,0],[9E9,9E9,9E9,9E9,9E9,9E9]];
            P03W13_Approach := [[0,0,0],[1,0,0,0],[0,0,0,0],[9E9,9E9,9E9,9E9,9E9,9E9]];
            P03W13_Retract := [[0,0,0],[1,0,0,0],[0,0,0,0],[9E9,9E9,9E9,9E9,9E9,9E9]];
            P03W13_Trans := [[0,0,0],[1,0,0,0],[0,0,0,0],[9E9,9E9,9E9,9E9,9E9,9E9]];
        ELSEIF slot = 14 THEN
            P03W14_Used := FALSE;
            P03W14_SubType := 0;
            P03W14_ToolSel := 0;
            P03W14_LenMM := 0;
            P03W14_ArcStart := [[0,0,0],[1,0,0,0],[0,0,0,0],[9E9,9E9,9E9,9E9,9E9,9E9]];
            P03W14_ArcEnd := [[0,0,0],[1,0,0,0],[0,0,0,0],[9E9,9E9,9E9,9E9,9E9,9E9]];
            P03W14_Approach := [[0,0,0],[1,0,0,0],[0,0,0,0],[9E9,9E9,9E9,9E9,9E9,9E9]];
            P03W14_Retract := [[0,0,0],[1,0,0,0],[0,0,0,0],[9E9,9E9,9E9,9E9,9E9,9E9]];
            P03W14_Trans := [[0,0,0],[1,0,0,0],[0,0,0,0],[9E9,9E9,9E9,9E9,9E9,9E9]];
        ELSEIF slot = 15 THEN
            P03W15_Used := FALSE;
            P03W15_SubType := 0;
            P03W15_ToolSel := 0;
            P03W15_LenMM := 0;
            P03W15_ArcStart := [[0,0,0],[1,0,0,0],[0,0,0,0],[9E9,9E9,9E9,9E9,9E9,9E9]];
            P03W15_ArcEnd := [[0,0,0],[1,0,0,0],[0,0,0,0],[9E9,9E9,9E9,9E9,9E9,9E9]];
            P03W15_Approach := [[0,0,0],[1,0,0,0],[0,0,0,0],[9E9,9E9,9E9,9E9,9E9,9E9]];
            P03W15_Retract := [[0,0,0],[1,0,0,0],[0,0,0,0],[9E9,9E9,9E9,9E9,9E9,9E9]];
            P03W15_Trans := [[0,0,0],[1,0,0,0],[0,0,0,0],[9E9,9E9,9E9,9E9,9E9,9E9]];
        ELSEIF slot = 16 THEN
            P03W16_Used := FALSE;
            P03W16_SubType := 0;
            P03W16_ToolSel := 0;
            P03W16_LenMM := 0;
            P03W16_ArcStart := [[0,0,0],[1,0,0,0],[0,0,0,0],[9E9,9E9,9E9,9E9,9E9,9E9]];
            P03W16_ArcEnd := [[0,0,0],[1,0,0,0],[0,0,0,0],[9E9,9E9,9E9,9E9,9E9,9E9]];
            P03W16_Approach := [[0,0,0],[1,0,0,0],[0,0,0,0],[9E9,9E9,9E9,9E9,9E9,9E9]];
            P03W16_Retract := [[0,0,0],[1,0,0,0],[0,0,0,0],[9E9,9E9,9E9,9E9,9E9,9E9]];
            P03W16_Trans := [[0,0,0],[1,0,0,0],[0,0,0,0],[9E9,9E9,9E9,9E9,9E9,9E9]];
        ELSEIF slot = 17 THEN
            P03W17_Used := FALSE;
            P03W17_SubType := 0;
            P03W17_ToolSel := 0;
            P03W17_LenMM := 0;
            P03W17_ArcStart := [[0,0,0],[1,0,0,0],[0,0,0,0],[9E9,9E9,9E9,9E9,9E9,9E9]];
            P03W17_ArcEnd := [[0,0,0],[1,0,0,0],[0,0,0,0],[9E9,9E9,9E9,9E9,9E9,9E9]];
            P03W17_Approach := [[0,0,0],[1,0,0,0],[0,0,0,0],[9E9,9E9,9E9,9E9,9E9,9E9]];
            P03W17_Retract := [[0,0,0],[1,0,0,0],[0,0,0,0],[9E9,9E9,9E9,9E9,9E9,9E9]];
            P03W17_Trans := [[0,0,0],[1,0,0,0],[0,0,0,0],[9E9,9E9,9E9,9E9,9E9,9E9]];
        ELSEIF slot = 18 THEN
            P03W18_Used := FALSE;
            P03W18_SubType := 0;
            P03W18_ToolSel := 0;
            P03W18_LenMM := 0;
            P03W18_ArcStart := [[0,0,0],[1,0,0,0],[0,0,0,0],[9E9,9E9,9E9,9E9,9E9,9E9]];
            P03W18_ArcEnd := [[0,0,0],[1,0,0,0],[0,0,0,0],[9E9,9E9,9E9,9E9,9E9,9E9]];
            P03W18_Approach := [[0,0,0],[1,0,0,0],[0,0,0,0],[9E9,9E9,9E9,9E9,9E9,9E9]];
            P03W18_Retract := [[0,0,0],[1,0,0,0],[0,0,0,0],[9E9,9E9,9E9,9E9,9E9,9E9]];
            P03W18_Trans := [[0,0,0],[1,0,0,0],[0,0,0,0],[9E9,9E9,9E9,9E9,9E9,9E9]];
        ELSEIF slot = 19 THEN
            P03W19_Used := FALSE;
            P03W19_SubType := 0;
            P03W19_ToolSel := 0;
            P03W19_LenMM := 0;
            P03W19_ArcStart := [[0,0,0],[1,0,0,0],[0,0,0,0],[9E9,9E9,9E9,9E9,9E9,9E9]];
            P03W19_ArcEnd := [[0,0,0],[1,0,0,0],[0,0,0,0],[9E9,9E9,9E9,9E9,9E9,9E9]];
            P03W19_Approach := [[0,0,0],[1,0,0,0],[0,0,0,0],[9E9,9E9,9E9,9E9,9E9,9E9]];
            P03W19_Retract := [[0,0,0],[1,0,0,0],[0,0,0,0],[9E9,9E9,9E9,9E9,9E9,9E9]];
            P03W19_Trans := [[0,0,0],[1,0,0,0],[0,0,0,0],[9E9,9E9,9E9,9E9,9E9,9E9]];
        ELSEIF slot = 20 THEN
            P03W20_Used := FALSE;
            P03W20_SubType := 0;
            P03W20_ToolSel := 0;
            P03W20_LenMM := 0;
            P03W20_ArcStart := [[0,0,0],[1,0,0,0],[0,0,0,0],[9E9,9E9,9E9,9E9,9E9,9E9]];
            P03W20_ArcEnd := [[0,0,0],[1,0,0,0],[0,0,0,0],[9E9,9E9,9E9,9E9,9E9,9E9]];
            P03W20_Approach := [[0,0,0],[1,0,0,0],[0,0,0,0],[9E9,9E9,9E9,9E9,9E9,9E9]];
            P03W20_Retract := [[0,0,0],[1,0,0,0],[0,0,0,0],[9E9,9E9,9E9,9E9,9E9,9E9]];
            P03W20_Trans := [[0,0,0],[1,0,0,0],[0,0,0,0],[9E9,9E9,9E9,9E9,9E9,9E9]];
        ELSEIF slot = 21 THEN
            P03W21_Used := FALSE;
            P03W21_SubType := 0;
            P03W21_ToolSel := 0;
            P03W21_LenMM := 0;
            P03W21_ArcStart := [[0,0,0],[1,0,0,0],[0,0,0,0],[9E9,9E9,9E9,9E9,9E9,9E9]];
            P03W21_ArcEnd := [[0,0,0],[1,0,0,0],[0,0,0,0],[9E9,9E9,9E9,9E9,9E9,9E9]];
            P03W21_Approach := [[0,0,0],[1,0,0,0],[0,0,0,0],[9E9,9E9,9E9,9E9,9E9,9E9]];
            P03W21_Retract := [[0,0,0],[1,0,0,0],[0,0,0,0],[9E9,9E9,9E9,9E9,9E9,9E9]];
            P03W21_Trans := [[0,0,0],[1,0,0,0],[0,0,0,0],[9E9,9E9,9E9,9E9,9E9,9E9]];
        ELSEIF slot = 22 THEN
            P03W22_Used := FALSE;
            P03W22_SubType := 0;
            P03W22_ToolSel := 0;
            P03W22_LenMM := 0;
            P03W22_ArcStart := [[0,0,0],[1,0,0,0],[0,0,0,0],[9E9,9E9,9E9,9E9,9E9,9E9]];
            P03W22_ArcEnd := [[0,0,0],[1,0,0,0],[0,0,0,0],[9E9,9E9,9E9,9E9,9E9,9E9]];
            P03W22_Approach := [[0,0,0],[1,0,0,0],[0,0,0,0],[9E9,9E9,9E9,9E9,9E9,9E9]];
            P03W22_Retract := [[0,0,0],[1,0,0,0],[0,0,0,0],[9E9,9E9,9E9,9E9,9E9,9E9]];
            P03W22_Trans := [[0,0,0],[1,0,0,0],[0,0,0,0],[9E9,9E9,9E9,9E9,9E9,9E9]];
        ELSEIF slot = 23 THEN
            P03W23_Used := FALSE;
            P03W23_SubType := 0;
            P03W23_ToolSel := 0;
            P03W23_LenMM := 0;
            P03W23_ArcStart := [[0,0,0],[1,0,0,0],[0,0,0,0],[9E9,9E9,9E9,9E9,9E9,9E9]];
            P03W23_ArcEnd := [[0,0,0],[1,0,0,0],[0,0,0,0],[9E9,9E9,9E9,9E9,9E9,9E9]];
            P03W23_Approach := [[0,0,0],[1,0,0,0],[0,0,0,0],[9E9,9E9,9E9,9E9,9E9,9E9]];
            P03W23_Retract := [[0,0,0],[1,0,0,0],[0,0,0,0],[9E9,9E9,9E9,9E9,9E9,9E9]];
            P03W23_Trans := [[0,0,0],[1,0,0,0],[0,0,0,0],[9E9,9E9,9E9,9E9,9E9,9E9]];
        ELSEIF slot = 24 THEN
            P03W24_Used := FALSE;
            P03W24_SubType := 0;
            P03W24_ToolSel := 0;
            P03W24_LenMM := 0;
            P03W24_ArcStart := [[0,0,0],[1,0,0,0],[0,0,0,0],[9E9,9E9,9E9,9E9,9E9,9E9]];
            P03W24_ArcEnd := [[0,0,0],[1,0,0,0],[0,0,0,0],[9E9,9E9,9E9,9E9,9E9,9E9]];
            P03W24_Approach := [[0,0,0],[1,0,0,0],[0,0,0,0],[9E9,9E9,9E9,9E9,9E9,9E9]];
            P03W24_Retract := [[0,0,0],[1,0,0,0],[0,0,0,0],[9E9,9E9,9E9,9E9,9E9,9E9]];
            P03W24_Trans := [[0,0,0],[1,0,0,0],[0,0,0,0],[9E9,9E9,9E9,9E9,9E9,9E9]];
        ELSEIF slot = 25 THEN
            P03W25_Used := FALSE;
            P03W25_SubType := 0;
            P03W25_ToolSel := 0;
            P03W25_LenMM := 0;
            P03W25_ArcStart := [[0,0,0],[1,0,0,0],[0,0,0,0],[9E9,9E9,9E9,9E9,9E9,9E9]];
            P03W25_ArcEnd := [[0,0,0],[1,0,0,0],[0,0,0,0],[9E9,9E9,9E9,9E9,9E9,9E9]];
            P03W25_Approach := [[0,0,0],[1,0,0,0],[0,0,0,0],[9E9,9E9,9E9,9E9,9E9,9E9]];
            P03W25_Retract := [[0,0,0],[1,0,0,0],[0,0,0,0],[9E9,9E9,9E9,9E9,9E9,9E9]];
            P03W25_Trans := [[0,0,0],[1,0,0,0],[0,0,0,0],[9E9,9E9,9E9,9E9,9E9,9E9]];
        ELSEIF slot = 26 THEN
            P03W26_Used := FALSE;
            P03W26_SubType := 0;
            P03W26_ToolSel := 0;
            P03W26_LenMM := 0;
            P03W26_ArcStart := [[0,0,0],[1,0,0,0],[0,0,0,0],[9E9,9E9,9E9,9E9,9E9,9E9]];
            P03W26_ArcEnd := [[0,0,0],[1,0,0,0],[0,0,0,0],[9E9,9E9,9E9,9E9,9E9,9E9]];
            P03W26_Approach := [[0,0,0],[1,0,0,0],[0,0,0,0],[9E9,9E9,9E9,9E9,9E9,9E9]];
            P03W26_Retract := [[0,0,0],[1,0,0,0],[0,0,0,0],[9E9,9E9,9E9,9E9,9E9,9E9]];
            P03W26_Trans := [[0,0,0],[1,0,0,0],[0,0,0,0],[9E9,9E9,9E9,9E9,9E9,9E9]];
        ELSEIF slot = 27 THEN
            P03W27_Used := FALSE;
            P03W27_SubType := 0;
            P03W27_ToolSel := 0;
            P03W27_LenMM := 0;
            P03W27_ArcStart := [[0,0,0],[1,0,0,0],[0,0,0,0],[9E9,9E9,9E9,9E9,9E9,9E9]];
            P03W27_ArcEnd := [[0,0,0],[1,0,0,0],[0,0,0,0],[9E9,9E9,9E9,9E9,9E9,9E9]];
            P03W27_Approach := [[0,0,0],[1,0,0,0],[0,0,0,0],[9E9,9E9,9E9,9E9,9E9,9E9]];
            P03W27_Retract := [[0,0,0],[1,0,0,0],[0,0,0,0],[9E9,9E9,9E9,9E9,9E9,9E9]];
            P03W27_Trans := [[0,0,0],[1,0,0,0],[0,0,0,0],[9E9,9E9,9E9,9E9,9E9,9E9]];
        ELSEIF slot = 28 THEN
            P03W28_Used := FALSE;
            P03W28_SubType := 0;
            P03W28_ToolSel := 0;
            P03W28_LenMM := 0;
            P03W28_ArcStart := [[0,0,0],[1,0,0,0],[0,0,0,0],[9E9,9E9,9E9,9E9,9E9,9E9]];
            P03W28_ArcEnd := [[0,0,0],[1,0,0,0],[0,0,0,0],[9E9,9E9,9E9,9E9,9E9,9E9]];
            P03W28_Approach := [[0,0,0],[1,0,0,0],[0,0,0,0],[9E9,9E9,9E9,9E9,9E9,9E9]];
            P03W28_Retract := [[0,0,0],[1,0,0,0],[0,0,0,0],[9E9,9E9,9E9,9E9,9E9,9E9]];
            P03W28_Trans := [[0,0,0],[1,0,0,0],[0,0,0,0],[9E9,9E9,9E9,9E9,9E9,9E9]];
        ELSEIF slot = 29 THEN
            P03W29_Used := FALSE;
            P03W29_SubType := 0;
            P03W29_ToolSel := 0;
            P03W29_LenMM := 0;
            P03W29_ArcStart := [[0,0,0],[1,0,0,0],[0,0,0,0],[9E9,9E9,9E9,9E9,9E9,9E9]];
            P03W29_ArcEnd := [[0,0,0],[1,0,0,0],[0,0,0,0],[9E9,9E9,9E9,9E9,9E9,9E9]];
            P03W29_Approach := [[0,0,0],[1,0,0,0],[0,0,0,0],[9E9,9E9,9E9,9E9,9E9,9E9]];
            P03W29_Retract := [[0,0,0],[1,0,0,0],[0,0,0,0],[9E9,9E9,9E9,9E9,9E9,9E9]];
            P03W29_Trans := [[0,0,0],[1,0,0,0],[0,0,0,0],[9E9,9E9,9E9,9E9,9E9,9E9]];
        ELSEIF slot = 30 THEN
            P03W30_Used := FALSE;
            P03W30_SubType := 0;
            P03W30_ToolSel := 0;
            P03W30_LenMM := 0;
            P03W30_ArcStart := [[0,0,0],[1,0,0,0],[0,0,0,0],[9E9,9E9,9E9,9E9,9E9,9E9]];
            P03W30_ArcEnd := [[0,0,0],[1,0,0,0],[0,0,0,0],[9E9,9E9,9E9,9E9,9E9,9E9]];
            P03W30_Approach := [[0,0,0],[1,0,0,0],[0,0,0,0],[9E9,9E9,9E9,9E9,9E9,9E9]];
            P03W30_Retract := [[0,0,0],[1,0,0,0],[0,0,0,0],[9E9,9E9,9E9,9E9,9E9,9E9]];
            P03W30_Trans := [[0,0,0],[1,0,0,0],[0,0,0,0],[9E9,9E9,9E9,9E9,9E9,9E9]];
        ELSE
            TPWrite "Invalid weld slot.";
        ENDIF
    ENDPROC

    PROC StoreNextFree_P03(num subType, num toolSel, num lenMM,
                       robtarget arcStart, robtarget arcEnd, robtarget approach, robtarget retract, robtarget trans)
        IF NOT P03W01_Used THEN
            StoreSlot_P03 1, subType, toolSel, lenMM, arcStart, arcEnd, approach, retract, trans;
            nWeldsP03 := nWeldsP03 + 1;
            RETURN;
        ELSEIF NOT P03W02_Used THEN
            StoreSlot_P03 2, subType, toolSel, lenMM, arcStart, arcEnd, approach, retract, trans;
            nWeldsP03 := nWeldsP03 + 1;
            RETURN;
        ELSEIF NOT P03W03_Used THEN
            StoreSlot_P03 3, subType, toolSel, lenMM, arcStart, arcEnd, approach, retract, trans;
            nWeldsP03 := nWeldsP03 + 1;
            RETURN;
        ELSEIF NOT P03W04_Used THEN
            StoreSlot_P03 4, subType, toolSel, lenMM, arcStart, arcEnd, approach, retract, trans;
            nWeldsP03 := nWeldsP03 + 1;
            RETURN;
        ELSEIF NOT P03W05_Used THEN
            StoreSlot_P03 5, subType, toolSel, lenMM, arcStart, arcEnd, approach, retract, trans;
            nWeldsP03 := nWeldsP03 + 1;
            RETURN;
        ELSEIF NOT P03W06_Used THEN
            StoreSlot_P03 6, subType, toolSel, lenMM, arcStart, arcEnd, approach, retract, trans;
            nWeldsP03 := nWeldsP03 + 1;
            RETURN;
        ELSEIF NOT P03W07_Used THEN
            StoreSlot_P03 7, subType, toolSel, lenMM, arcStart, arcEnd, approach, retract, trans;
            nWeldsP03 := nWeldsP03 + 1;
            RETURN;
        ELSEIF NOT P03W08_Used THEN
            StoreSlot_P03 8, subType, toolSel, lenMM, arcStart, arcEnd, approach, retract, trans;
            nWeldsP03 := nWeldsP03 + 1;
            RETURN;
        ELSEIF NOT P03W09_Used THEN
            StoreSlot_P03 9, subType, toolSel, lenMM, arcStart, arcEnd, approach, retract, trans;
            nWeldsP03 := nWeldsP03 + 1;
            RETURN;
        ELSEIF NOT P03W10_Used THEN
            StoreSlot_P03 10, subType, toolSel, lenMM, arcStart, arcEnd, approach, retract, trans;
            nWeldsP03 := nWeldsP03 + 1;
            RETURN;
        ELSEIF NOT P03W11_Used THEN
            StoreSlot_P03 11, subType, toolSel, lenMM, arcStart, arcEnd, approach, retract, trans;
            nWeldsP03 := nWeldsP03 + 1;
            RETURN;
        ELSEIF NOT P03W12_Used THEN
            StoreSlot_P03 12, subType, toolSel, lenMM, arcStart, arcEnd, approach, retract, trans;
            nWeldsP03 := nWeldsP03 + 1;
            RETURN;
        ELSEIF NOT P03W13_Used THEN
            StoreSlot_P03 13, subType, toolSel, lenMM, arcStart, arcEnd, approach, retract, trans;
            nWeldsP03 := nWeldsP03 + 1;
            RETURN;
        ELSEIF NOT P03W14_Used THEN
            StoreSlot_P03 14, subType, toolSel, lenMM, arcStart, arcEnd, approach, retract, trans;
            nWeldsP03 := nWeldsP03 + 1;
            RETURN;
        ELSEIF NOT P03W15_Used THEN
            StoreSlot_P03 15, subType, toolSel, lenMM, arcStart, arcEnd, approach, retract, trans;
            nWeldsP03 := nWeldsP03 + 1;
            RETURN;
        ELSEIF NOT P03W16_Used THEN
            StoreSlot_P03 16, subType, toolSel, lenMM, arcStart, arcEnd, approach, retract, trans;
            nWeldsP03 := nWeldsP03 + 1;
            RETURN;
        ELSEIF NOT P03W17_Used THEN
            StoreSlot_P03 17, subType, toolSel, lenMM, arcStart, arcEnd, approach, retract, trans;
            nWeldsP03 := nWeldsP03 + 1;
            RETURN;
        ELSEIF NOT P03W18_Used THEN
            StoreSlot_P03 18, subType, toolSel, lenMM, arcStart, arcEnd, approach, retract, trans;
            nWeldsP03 := nWeldsP03 + 1;
            RETURN;
        ELSEIF NOT P03W19_Used THEN
            StoreSlot_P03 19, subType, toolSel, lenMM, arcStart, arcEnd, approach, retract, trans;
            nWeldsP03 := nWeldsP03 + 1;
            RETURN;
        ELSEIF NOT P03W20_Used THEN
            StoreSlot_P03 20, subType, toolSel, lenMM, arcStart, arcEnd, approach, retract, trans;
            nWeldsP03 := nWeldsP03 + 1;
            RETURN;
        ELSEIF NOT P03W21_Used THEN
            StoreSlot_P03 21, subType, toolSel, lenMM, arcStart, arcEnd, approach, retract, trans;
            nWeldsP03 := nWeldsP03 + 1;
            RETURN;
        ELSEIF NOT P03W22_Used THEN
            StoreSlot_P03 22, subType, toolSel, lenMM, arcStart, arcEnd, approach, retract, trans;
            nWeldsP03 := nWeldsP03 + 1;
            RETURN;
        ELSEIF NOT P03W23_Used THEN
            StoreSlot_P03 23, subType, toolSel, lenMM, arcStart, arcEnd, approach, retract, trans;
            nWeldsP03 := nWeldsP03 + 1;
            RETURN;
        ELSEIF NOT P03W24_Used THEN
            StoreSlot_P03 24, subType, toolSel, lenMM, arcStart, arcEnd, approach, retract, trans;
            nWeldsP03 := nWeldsP03 + 1;
            RETURN;
        ELSEIF NOT P03W25_Used THEN
            StoreSlot_P03 25, subType, toolSel, lenMM, arcStart, arcEnd, approach, retract, trans;
            nWeldsP03 := nWeldsP03 + 1;
            RETURN;
        ELSEIF NOT P03W26_Used THEN
            StoreSlot_P03 26, subType, toolSel, lenMM, arcStart, arcEnd, approach, retract, trans;
            nWeldsP03 := nWeldsP03 + 1;
            RETURN;
        ELSEIF NOT P03W27_Used THEN
            StoreSlot_P03 27, subType, toolSel, lenMM, arcStart, arcEnd, approach, retract, trans;
            nWeldsP03 := nWeldsP03 + 1;
            RETURN;
        ELSEIF NOT P03W28_Used THEN
            StoreSlot_P03 28, subType, toolSel, lenMM, arcStart, arcEnd, approach, retract, trans;
            nWeldsP03 := nWeldsP03 + 1;
            RETURN;
        ELSEIF NOT P03W29_Used THEN
            StoreSlot_P03 29, subType, toolSel, lenMM, arcStart, arcEnd, approach, retract, trans;
            nWeldsP03 := nWeldsP03 + 1;
            RETURN;
        ELSEIF NOT P03W30_Used THEN
            StoreSlot_P03 30, subType, toolSel, lenMM, arcStart, arcEnd, approach, retract, trans;
            nWeldsP03 := nWeldsP03 + 1;
            RETURN;
        ELSE
            TPWrite "No free weld slots available.";
        ENDIF
    ENDPROC

